// TwinCAT 3 PLC project TwinCore
// Title: TwinCore
// Company: TwinCore
// Author: TwinCore
// ProjectVersion: 2026.24.1.0
// Description: base implementations, utilities, TC3 event logging, state machines, ...
// ProgramVersion: 3.1.4026.23
// libraries:
//   Tc2_Standard, * (Beckhoff Automation GmbH)
//   Tc2_System, * (Beckhoff Automation GmbH)
//   Tc2_Utilities, * (Beckhoff Automation GmbH)
//   Tc3_EventLogger, * (Beckhoff Automation GmbH)
//   Tc3_Module, * (Beckhoff Automation GmbH)
// project tree:
//   EventLogger/EventListenerExtV2/DUTs/ E_AlarmMessage.TcDUT, ST_AlarmInfo.TcDUT, ST_AlarmLog.TcDUT, ST_EventEntryTableListener.TcDUT
//   EventLogger/EventListenerExtV2/ FB_EventListenerExtV2.TcPOU, I_EventListener.TcIO
//   EventLogger/EventManagement/DUTs/ E_AlarmReaction.TcDUT, ST_EventEntryTable.TcDUT, ST_EventHmiControl.TcDUT
//   EventLogger/EventManagement/ FB_Alarm.TcPOU, FB_AlarmDelayed.TcPOU, FB_AlarmManagement.TcPOU, FB_Message.TcPOU, I_Alarm.TcIO, I_Message.TcIO
//   EventLogger/Logger/ E_RollingInterval.TcDUT, FB_FileRetentionTimeHandler.TcPOU, FB_GenerateTimeData.TcPOU, FB_Log.TcPOU, FB_LogFile.TcPOU, FB_LogStringBuffer.TcPOU, FB_SystemTimeService.TcPOU, F_GetFileAgeInSeconds.TcPOU, ST_LogEntry.TcDUT
//   General/Blinker/ FB_Blinker.TcPOU, FB_Blinker_PWM.TcPOU
//   General/CONCAT/ FB_CONCAT.TcPOU, FB_CONCAT_STRINGS.TcPOU, I_CONCAT.TcIO
//   General/ FB_AnalogInputFilter.TcPOU, FB_Signal.TcPOU
//   GVLs/ GVL_Diag.TcGVL, GVL_GLOBAL.TcGVL
//   Lists/ FB_ListNumbers_DINT.TcPOU, FB_ListNumbers_REAL.TcPOU, FB_ListString.TcPOU
//   Misc/ ST_LinCoord_XY.TcDUT, ST_LinCoord_XYZ.TcDUT, ST_SysTime.TcDUT
//   / Parameter.TcGVL
//   Process/DUTs/ ST_Position.TcDUT, ST_ProcessData.TcDUT, ST_Task.TcDUT
//   Process/ FB_Process.TcPOU
//   Project Information/ F_GetCompany.TcPOU, F_GetTitle.TcPOU, F_GetVersion.TcPOU
//   StateMachine/ FB_StateMachine.TcPOU, ST_HMI_Condition.TcDUT, ST_HMI_StateMachine.TcDUT, ST_StateMachine_State.TcDUT
//   StateMachine/MachineState/ E_MachineState.TcDUT, FB_MachineState.TcPOU, ST_MachineInfo.TcDUT
//   StateMachine/ModeControl/ E_Mode.TcDUT, FB_ModeControl.TcPOU
//   Version/ Global_Version.TcGVL

// ---- EventLogger/EventListenerExtV2/DUTs/E_AlarmMessage.TcDUT
{attribute 'qualified_only'}
{attribute 'strict'}
TYPE E_AlarmMessage :
(
	RequestText := 0,
    ReceiveText := 1,
    Insert := 2,
    WriteDB := 3,
    Done := 4
);
END_TYPE

// ---- EventLogger/EventListenerExtV2/DUTs/ST_AlarmInfo.TcDUT
TYPE ST_AlarmInfo :
STRUCT
	bVerbose: BOOL;
	nVerboseRaisedCount: UDINT;
	bInfo: BOOL;
	nInfoRaisedCount: UDINT; 
	bWarning: BOOL;
	nWarningRaisedCount: UDINT;
	bError: BOOL;
	nErrorRaisedCount: UDINT;
	bCritical: BOOL;
	nCriticalRaisedCount: UDINT;
END_STRUCT
END_TYPE

// ---- EventLogger/EventListenerExtV2/DUTs/ST_AlarmLog.TcDUT
TYPE ST_AlarmLog :
STRUCT
	sTimestamp: STRING;
	sText: STRING(255); //
	sSourceName: STRING(255); //
	EventClassName: STRING(255); //
    eConfirmationState : INT;
    eSeverity :  INT; // INT
END_STRUCT
END_TYPE

// ---- EventLogger/EventListenerExtV2/DUTs/ST_EventEntryTableListener.TcDUT
TYPE ST_EventEntryTableListener EXTENDS ST_EventEntryTable:
STRUCT
	sJsonAttribute	: STRING(8000);
	ipArguments		: I_TcArguments;
END_STRUCT
END_TYPE

// ---- EventLogger/EventManagement/DUTs/E_AlarmReaction.TcDUT
{attribute 'qualified_only'}
{attribute 'strict'}
TYPE E_AlarmReaction :
(
	None := 0,
	Info,
	Warning,
	Verbose,
	StopAtCycleEnd,
	AbortGroup,
	AbortAll,
	MediaOff
);
END_TYPE

// ---- EventLogger/EventManagement/DUTs/ST_EventEntryTable.TcDUT
TYPE ST_EventEntryTable EXTENDS ST_LogEntry :
STRUCT
	nSourceId			: UDINT;
	nZoneId				: UDINT;
	nGroupId			: UDINT;
	sDescription		: T_MaxString;
	eSeverity			: TcEventSeverity;
	eReaction			: E_AlarmReaction;
    sReaction			: STRING( 24 );
	EventClass			: GUID;
	EventClassName		: T_MaxString;
	sTimestamp			: STRING( 24 );
	sTimestampConfirmed	: STRING( 24 );
	sTimestampCleared	: STRING( 24 );
	nEventId			: UDINT;
	eConfirmationState	: TcEventConfirmationState;
	bTextRecieved		: BOOL;
	bIsAlarm			: BOOL;
	bIsEvent			: BOOL;
    stAlarmLog			: ST_AlarmLog;
    bLogged				: BOOL;
    nLanguageId			: INT;
END_STRUCT
END_TYPE

// ---- EventLogger/EventManagement/DUTs/ST_EventHmiControl.TcDUT
TYPE ST_EventHmiControl :
STRUCT
END_STRUCT
END_TYPE

// ---- EventLogger/Logger/E_RollingInterval.TcDUT
{attribute 'qualified_only'}
{attribute 'strict'}
{attrivute 'to_string'}
// Rolling interval to create a new log file when expired. 
TYPE E_RollingInterval : (
    None,
    Hourly,
    Daily,
    Monthly
);
END_TYPE

// ---- EventLogger/Logger/ST_LogEntry.TcDUT
TYPE ST_LogEntry :
STRUCT
	sSeverity		:  STRING( 24 );
	sSourceName		: T_MaxString;
	sTimestampLog	: STRING( 24 );
	MethodName		: STRING( 24 );
	sText			: T_MaxString;
END_STRUCT
END_TYPE

// ---- Misc/ST_LinCoord_XY.TcDUT
TYPE ST_LinCoord_XY :
STRUCT
	x	: REAL;	// [mm]
	y	: REAL;	// [mm]
END_STRUCT
END_TYPE

// ---- Misc/ST_LinCoord_XYZ.TcDUT
TYPE ST_LinCoord_XYZ EXTENDS ST_LinCoord_XY :
STRUCT
	z	: REAL;	// [mm]
END_STRUCT
END_TYPE

// ---- Misc/ST_SysTime.TcDUT
TYPE ST_SysTime :
STRUCT
	uliDateTime	: ULINT := 0;
	sTimestamp	: STRING(12); // current time, format: hh:mm:ss:ms
	sDate		: STRING(10); // current date, format example: dd.mm.yyyy
	uiYear		: UINT := 0;
	uiMonth		: UINT := 9999;
	uiDay		: UINT := 9999;
	uiHour		: UINT := 9999;
	uiMinute	: UINT := 9999;
	uiSecond	: UINT := 9999;
	uiMillis	: UINT := 9999;
END_STRUCT
END_TYPE

// ---- Process/DUTs/ST_Position.TcDUT
TYPE ST_Position :
STRUCT
	Task		: ARRAY[0..Parameter.MAX_TASK_INDEX] OF ST_Task;
	Group		: ARRAY[0..Parameter.MAX_GROUP_INDEX] OF ST_Task;
	Info		: ST_Task;
END_STRUCT
END_TYPE

// ---- Process/DUTs/ST_ProcessData.TcDUT
TYPE ST_ProcessData :
STRUCT
	Pos	: ARRAY[0..Parameter.MAX_POS_INDEX] OF ST_Position;
	Info		: ST_Task;	// info about the complete process of all positions
END_STRUCT
END_TYPE

// ---- Process/DUTs/ST_Task.TcDUT
TYPE ST_Task :
STRUCT
	Enabled		: BOOL := FALSE;	// false if not existing
	Released	: BOOL;	// free to start this task
	Busy		: BOOL;	// task started
	Finished	: BOOL;	// also TRUE, when all Tasks are disabled
	OK			: BOOL;
	NOK			: BOOL;
	ManualOK	: BOOL;
	ManualNOK	: BOOL;
	State		: USINT;	// lamp HMI
	(*	State
		0 - not existing
		1 - existing/enabled, but not released
		2 - enabled and released, ready to process
		3 - processing, process started
		4 - OK
		5 - NOK
		6 - ManualOK
		7 - ManualNOK
	*)
	_groupID	: USINT := 0;
END_STRUCT
END_TYPE

// ---- StateMachine/MachineState/E_MachineState.TcDUT
{attribute 'qualified_only'}
TYPE E_MachineState :
(
	Error := -1,
	Idle := 0,
	Stopped,	// Manual Control
	Stopping,
	Aborting,
	Aborted,
	Starting,
	Execute,	// Automatic
	Hold,
	Homing,
	Clearing,
	Resetting
);
END_TYPE

// ---- StateMachine/MachineState/ST_MachineInfo.TcDUT
TYPE ST_MachineInfo :
STRUCT
	bInInitDone:	BOOL;
	bInMediaOn:		BOOL;
END_STRUCT
END_TYPE

// ---- StateMachine/ModeControl/E_Mode.TcDUT
{attribute 'qualified_only'}
TYPE E_Mode :
(
	Error := -1,
	Idle := 0,
	Stopped,	// Manual Control
	Stopping,
	Aborting,
	Aborted,
	Starting,
	Hold,
	Homing,
	Clearing,
	Resetting,
	Standby,	// Automatic
	Execute	// Automatic
);
END_TYPE

// ---- StateMachine/ST_HMI_Condition.TcDUT
TYPE ST_HMI_Condition :
STRUCT
	xState	: BOOL := TRUE;
	sName	: STRING(26) := '';
END_STRUCT
END_TYPE

// ---- StateMachine/ST_HMI_StateMachine.TcDUT
TYPE ST_HMI_StateMachine :
STRUCT
	// name of state machine
	sName				: STRING;	

	// current state
	nState				: INT;
	nNextState			: INT;	// prepared next state
	sState				: STRING;
	
	// conditions
	stSwitchCondition	: ARRAY[0..Parameter.NUM_CON] OF ST_HMI_Condition;
	stStateCondition	: ARRAY[0..Parameter.NUM_CON] OF ST_HMI_Condition;
	
	nSwitchOrSection	: INT;	// current or section
	bShowOrSection		: BOOL;	// show or section elements
	bShowNextState		: BOOL;	// show next state
	bSwitchOrSectionDec	: BOOL;	// decrement
	bSwitchOrSectionInc	: BOOL;	// increment
	bStepMode			: BOOL;
	bStepNext			: BOOL;
	
	// Log
	stStateHistory		: ARRAY[0..Parameter.HISTORY_SIZE] OF ST_StateMachine_State;
END_STRUCT
END_TYPE

// ---- StateMachine/ST_StateMachine_State.TcDUT
TYPE ST_StateMachine_State :
STRUCT
	nState	: INT;
	sState	: STRING;
END_STRUCT
END_TYPE

// ---- GVLs/GVL_Diag.TcGVL
{attribute 'qualified_only'}
VAR_GLOBAL
	gfbAlarmManagement			: FB_AlarmManagement;	// first: nested FB_Alarm.FB_init prepends onto ipAlarmHead
	gfbLogFile					: FB_LogFile;
	gfbEventListener			: FB_EventListenerExtV2; // other HMI than TE2000
	ipAlarmHead					: I_Alarm;	// singly linked list of all FB_Alarm instances
	gnCountAlarms				: UINT := 0;	// built-in and user FB_Alarm instances self-register in FB_init
	gbCountAlarmsMaxExceeded	: BOOL := FALSE;
	gbInterfaceNotAssigned		: BOOL := FALSE;
	
END_VAR

// ---- GVLs/GVL_GLOBAL.TcGVL
{attribute 'Tc2GvlVarNames'}
VAR_GLOBAL
	fbConcat		: FB_CONCAT;
    fbSystemTime	: FB_SystemTimeService;
END_VAR

// ---- Parameter.TcGVL
{attribute 'qualified_only'}
VAR_GLOBAL CONSTANT
	
    MAX_STRING_LENGTH	: UDINT := 255;
	
	
	// Alarm Management
	nMaxNumberAlarms		: UINT := 2000;	// safety cap for FB_Alarm linked-list registration (not an array size)
	
	// Logger
	MAX_LOG_STRING_SIZE		: UINT := 1000;	// maximal string size for one log entry (line)
    MAX_BUFFER_COUNT		: UDINT := 1000;
	
	// Following for other HMI solution than TE2000
	nMaxEventEntries		: UINT := 200;	// max. event entries in EventEntryTable
	
	// Listener
	nMaxEventClasses		: UINT := 2;	// Listener - max. event classes
	nNUM_OF_MESSAGES_VISU	: UINT := 15;	// Listener - messages to store and read from HMI
	
	
	// state machine
	NUM_CON			: USINT := 15;
	HISTORY_SIZE	: INT := 30;
	
	// Process
	MAX_POS_INDEX	: INT := 4;
	MAX_TASK_INDEX	: INT := 81;
	MAX_GROUP_INDEX	: INT := 15;
	
END_VAR

// ---- Version/Global_Version.TcGVL
{attribute 'TcGenerated'}
{attribute 'no-analysis'}
{attribute 'linkalways'}
// This function has been automatically generated from the project information.
VAR_GLOBAL CONSTANT
	{attribute 'const_non_replaced'}
	stLibVersion_TwinCore : ST_LibVersion := (iMajor := 2026, iMinor := 24, iBuild := 1, iRevision := 0, nFlags := 1, sVersion := '2026.24.1.0');
END_VAR

// ---- EventLogger/EventListenerExtV2/I_EventListener.TcIO
INTERFACE I_EventListener EXTENDS __SYSTEM.IQueryInterface

METHOD PUBLIC DeleteEventsFromTable : BOOL
END_METHOD

METHOD GetEventByIndex : HRESULT
    VAR_OUTPUT
        sTimestamp: STRING(80); // 
        sTimestampConfirmed: STRING(80);
        sTimestampCleared: STRING(80);
        sText: STRING(255); //
        sSourceName: STRING(255); //
        EventClassName: STRING(255); //
        eConfirmationState : BYTE;
        eSeverity :  BYTE; // INT
    END_VAR
VAR_INPUT
    nIndex : UDINT;
END_VAR
END_METHOD

PROPERTY PUBLIC LangId : INT
GET
END_GET
SET
END_SET
END_PROPERTY

PROPERTY NumberActiveEvents : UDINT
GET
END_GET
END_PROPERTY

END_INTERFACE

// ---- EventLogger/EventManagement/I_Alarm.TcIO
INTERFACE I_Alarm EXTENDS I_Message

METHOD Ack : HRESULT
VAR_INPUT
END_VAR
END_METHOD

PROPERTY bActive : BOOL
GET
END_GET
END_PROPERTY

PROPERTY PUBLIC bBlockAck : BOOL
GET
END_GET
SET
END_SET
END_PROPERTY

PROPERTY bRaised : BOOL
GET
END_GET
END_PROPERTY

PROPERTY PUBLIC eEventReaction : E_AlarmReaction
GET
END_GET
END_PROPERTY

PROPERTY ipNext : I_Alarm
GET
END_GET
SET
END_SET
END_PROPERTY

METHOD PUBLIC UpdateText : HRESULT
VAR_INPUT
	LangId	: INT;
END_VAR
END_METHOD

END_INTERFACE

// ---- EventLogger/EventManagement/I_Message.TcIO
 INTERFACE I_Message

PROPERTY PUBLIC bSetEvent : BOOL
GET
END_GET
SET
END_SET
END_PROPERTY

PROPERTY eSeverity : TcEventSeverity
GET
END_GET
END_PROPERTY

METHOD GetEventEntry : ST_EventEntryTable
VAR_INPUT
END_VAR
END_METHOD

METHOD GetEventText : BOOL
VAR_INPUT
END_VAR
END_METHOD

METHOD GetJsonAttribute : HRESULT
VAR_INPUT
	sJsonAttribute	: REFERENCE TO STRING;
	nJsonAttribute	: UDINT;
END_VAR
END_METHOD

PROPERTY PUBLIC LogEntry : ST_LogEntry
GET
END_GET
END_PROPERTY

PROPERTY PUBLIC nGetGroupId : UINT
GET
END_GET
END_PROPERTY

PROPERTY PUBLIC nGetSourceId : UDINT
GET
END_GET
END_PROPERTY

END_INTERFACE

// ---- General/CONCAT/I_CONCAT.TcIO
INTERFACE I_CONCAT

METHOD AddString : I_CONCAT
VAR_INPUT
	pSrcString	: ANY_STRING;
END_VAR
END_METHOD

METHOD AddStringInput : I_CONCAT
VAR_INPUT
	in:	STRING;
END_VAR
END_METHOD

METHOD PUBLIC Get : T_MAXSTRING
VAR_INPUT
END_VAR
END_METHOD

END_INTERFACE

// ---- EventLogger/EventManagement/FB_AlarmManagement.TcPOU
FUNCTION_BLOCK FB_AlarmManagement
VAR_INPUT
	bInAck			: BOOL;	// Acknowledge all errors, if possible
END_VAR
VAR_OUTPUT
	bError			: BOOL;	// Alarm active with reaction type media off or abort all
	
	// MessageReaction
	bVerbose		: BOOL;	// at least one verbose info is active (not important info)
	bInfo			: BOOL;	// at least one info is active
	bWarning		: BOOL;	// at least one warning is active
	bStopAtCycleEnd	: BOOL;	// at least on alarm needs to stop at cycle end, goes into stop state after ending cycle
	bAbortGroup		: BOOL;	// aborts one group, detect with method IsAlarmInGroup( GroupID ) or IsAlarmInGroupOfZone( GroupID )
	bAbortAll		: BOOL;	// abort/stops all groups
	bMediaOff		: BOOL;	// critical alarm, shuts down media!
	
	bAckRequested	: BOOL;	// at least one verbose info is active (not important info)
	
    aEventEntryTable: ARRAY[0..Parameter.nMaxEventEntries] OF ST_EventEntryTable;	// to show in HMI
	
END_VAR
VAR
	bInit	: BOOL := TRUE;
	
    nCounter	: UINT;

	rtAck	: R_TRIG;
	
	nVisuTableIndex					: UINT;
	bVisuTableCmdIndexPlus			: BOOL;
	bVisuTableCmdIndexMinus			: BOOL;
	bVisuTableDisableCmdIndexPlus	: BOOL;
	bVisuTableDisableCmdIndexMinus	: BOOL;
	bVisuTableCmdCleanErrors		: BOOL;
	
    nLanguage	: INT := 1031;
    sLanguage	: STRING := 'de';
    bChangeLanguage	: BOOL;
	
	cfgShowErrors	: BOOL := TRUE;	// including critical
	cfgShowWarnings	: BOOL := TRUE;
	cfgShowInfos	: BOOL := TRUE;	// including verbose
	
    fbSourceInfo				: FB_TcSourceInfo;
    fbGetTimeZoneInformation	: FB_GetTimeZoneInformation;
    stSeverestAlarmEntryTable	: ST_EventEntryTable;
    stLastEventEntryTable		: ST_EventEntryTable;
	
	fbWrnTooManyAlarms			: FB_Alarm( TC_EVENTS.EventClassGeneral.W_TooManyAlarmsDefined );
	fbErrInterfaceNotAssigned	: FB_Alarm( TC_EVENTS.EventClassGeneral.E_Debug );
	fbWrnArgumentBeforeInit		: FB_Alarm( TC_EVENTS.EventClassGeneral.W_ArgumentBeforeInit );
	fbWrnCyclicCallNotDetected	: FB_Alarm( TC_EVENTS.EventClassGeneral.W_CyclicCallNotDetected );
	{warning 'TODO: realize cyclic call detection'}
	
END_VAR


// in case you only want to call the body cyclic.
Execute( bInAck );

{warning 'TODO: log history of general events! Verbose/Debug'}

// cyclic call of Event Management, in case you don't want to use the FB-body!
METHOD PUBLIC Execute : HRESULT
VAR_INPUT
	bInAck			: BOOL;	// Acknowledge all errors, if possible
END_VAR
VAR_INST
    bGetTimeZone : BOOL := TRUE;
END_VAR

// inititalizing
IF bInit THEN
	Initialize();
END_IF

// trigger of inputs
rtAck( CLK := bInAck OR bVisuTableCmdCleanErrors );
bVisuTableCmdCleanErrors R= bVisuTableCmdCleanErrors;

// check if at least one Error is raised, and store alarm reaction type
initOutputs();

// Update Language
LanguageId( sLanguage );

// Update event table
UpdateEventTable();

// HMI
HMI();

fbGetTimeZoneInformation( bExecute := bGetTimeZone );
bGetTimeZone R= bGetTimeZone;

// Debug Meldungen 
fbWrnTooManyAlarms.setEvent( GVL_Diag.gbCountAlarmsMaxExceeded );
fbErrInterfaceNotAssigned.setEvent( GVL_Diag.gbInterfaceNotAssigned );
fbWrnArgumentBeforeInit.setEvent( FALSE );
END_METHOD

METHOD FB_exit : BOOL
VAR_INPUT
	bInCopyCode : BOOL; // if TRUE, the exit method is called for exiting an instance that is copied afterwards (online change).
END_VAR

IF NOT bInCopyCode THEN
	; // each nested FB_Alarm.FB_exit unlinks itself from ipAlarmHead
END_IF
END_METHOD

METHOD PUBLIC GetEventTable : BOOL
VAR_INPUT
	nZoneId		: UDINT;	// Zone = 0 is for all zones
	nGroupId	: UINT;
	bShowError	: BOOL;	// including criticals
	bShowWarning: BOOL;
	bShowInfo	: BOOL;	// including verbose
END_VAR
VAR_IN_OUT
	astEventTable	:	ARRAY[*] OF ST_EventEntryTable;
END_VAR
VAR
	i			: DINT;
	j			: DINT;
	nLowerBound	: DINT;
	nUpperBound	: DINT;
	EmptyEventTableLine	: ST_EventEntryTable;
END_VAR

// check bounds
nLowerBound := LOWER_BOUND( astEventTable, 1 );
nUpperBound := UPPER_BOUND( astEventTable, 1 );
j := nLowerBound;

// empty table
FOR i := nLowerBound TO nUpperBound DO	
	astEventTable[i] := EmptyEventTableLine;
END_FOR

// poll the big Event table
FOR i := 0 TO Parameter.nMaxEventEntries DO

	// check filter settings
	IF ( nZoneId <> 0 AND aEventEntryTable[i].nZoneId = nZoneId )
	OR_ELSE ( nGroupId <> 0 AND aEventEntryTable[i].nGroupId = nGroupId )
	AND_THEN ( ( aEventEntryTable[i].eSeverity = TcEventSeverity.Critical AND bShowError )
		OR ( aEventEntryTable[i].eSeverity = TcEventSeverity.Error AND bShowError )
		OR ( aEventEntryTable[i].eSeverity = TcEventSeverity.Warning AND bShowWarning )
		OR ( aEventEntryTable[i].eSeverity = TcEventSeverity.Info AND bShowInfo )
		OR ( aEventEntryTable[i].eSeverity = TcEventSeverity.Verbose AND bShowInfo ) )
	THEN
		
		// fill filtered feedback table
		astEventTable[j] := aEventEntryTable[i];
		j := j + 1;
		
	END_IF
	
	// used table is full
	IF j > nUpperBound THEN
		RETURN;
	END_IF
	
END_FOR
END_METHOD

METHOD PRIVATE HMI : BOOL
VAR_INST
    nCounterTemp : DINT;
    trigVisuIndexingPlus: R_TRIG;
	trigVisuIndexingMinus: R_TRIG;
END_VAR

IF nCounterTemp <> nCounter THEN
    nCounterTemp := nCounter;
    nVisuTableIndex := 0;
END_IF

bVisuTableDisableCmdIndexPlus := nVisuTableIndex > nCounter - Parameter.nNUM_OF_MESSAGES_VISU
	OR nCounter <= Parameter.nNUM_OF_MESSAGES_VISU
	OR nVisuTableIndex >= Parameter.nMaxEventEntries;

bVisuTableDisableCmdIndexMinus := nVisuTableIndex <= 0;

trigVisuIndexingPlus( CLK := bVisuTableCmdIndexPlus );
IF trigVisuIndexingPlus.Q THEN
	nVisuTableIndex := nVisuTableIndex + 1;
END_IF

trigVisuIndexingMinus( CLK := bVisuTableCmdIndexMinus );
IF trigVisuIndexingMinus.Q THEN
	nVisuTableIndex := nVisuTableIndex - 1;
END_IF
END_METHOD

METHOD PRIVATE Initialize : BOOL
VAR_INPUT
END_VAR

fbWrnTooManyAlarms.Initialize( 0, 0, E_AlarmReaction.Warning );
fbErrInterfaceNotAssigned.Initialize( 0, 0, E_AlarmReaction.AbortAll );
fbWrnArgumentBeforeInit.Initialize( 0, 0, E_AlarmReaction.Warning );

bInit := FALSE;
END_METHOD

METHOD PRIVATE initOutputs : BOOL
VAR_INPUT
END_VAR

bError			:= FALSE;
bInfo			:= FALSE;
bWarning		:= FALSE;
bVerbose		:= FALSE;
bStopAtCycleEnd	:= FALSE;
bAbortGroup		:= FALSE;
bAbortAll		:= FALSE;
bMediaOff		:= FALSE;
END_METHOD

METHOD PUBLIC IsAlarmInGroup : BOOL
VAR_INPUT
	nGroupId	: UINT;
END_VAR
VAR
	ipAlarm	: I_Alarm;
	nGuard	: UINT;
END_VAR

IsAlarmInGroup := FALSE;
ipAlarm := GVL_Diag.ipAlarmHead;
nGuard := 0;
WHILE ipAlarm <> 0 AND nGuard < Parameter.nMaxNumberAlarms DO
	nGuard := nGuard + 1;
	IF ipAlarm.bActive
	AND_THEN ipAlarm.nGetGroupId = nGroupId THEN
		IsAlarmInGroup := TRUE;
		RETURN;
	END_IF
	ipAlarm := ipAlarm.ipNext;
END_WHILE
END_METHOD

METHOD PUBLIC IsAlarmInGroupOfZone : BOOL
VAR_INPUT
	nZoneId		: UDINT;
	nGroupId	: UINT;
END_VAR
VAR
	ipAlarm	: I_Alarm;
	nGuard	: UINT;
END_VAR

IsAlarmInGroupOfZone := FALSE;
ipAlarm := GVL_Diag.ipAlarmHead;
nGuard := 0;
WHILE ipAlarm <> 0 AND nGuard < Parameter.nMaxNumberAlarms DO
	nGuard := nGuard + 1;
	IF ipAlarm.bActive
	AND_THEN ipAlarm.nGetGroupId = nGroupId
	AND ipAlarm.nGetSourceId = nZoneId THEN
		IsAlarmInGroupOfZone := TRUE;
		RETURN;
	END_IF
	ipAlarm := ipAlarm.ipNext;
END_WHILE
END_METHOD

METHOD PUBLIC IsAlarmInZone : BOOL
VAR_INPUT
	nZoneId	: UDINT;
END_VAR
VAR
	ipAlarm	: I_Alarm;
	nGuard	: UINT;
END_VAR

IsAlarmInZone := FALSE;
ipAlarm := GVL_Diag.ipAlarmHead;
nGuard := 0;
WHILE ipAlarm <> 0 AND nGuard < Parameter.nMaxNumberAlarms DO
	nGuard := nGuard + 1;
	IF ipAlarm.bActive
	AND_THEN ipAlarm.nGetSourceId = nZoneId THEN
		IsAlarmInZone := TRUE;
		RETURN;
	END_IF
	ipAlarm := ipAlarm.ipNext;
END_WHILE
END_METHOD

METHOD PUBLIC LanguageId : HRESULT
VAR_INPUT
	sCurrentLanguage	: STRING;
END_VAR
VAR
	ipAlarm	: I_Alarm;
	nGuard	: UINT;
	hrChangeLang	:HRESULT;
	bChangeLangPending	:BOOL;
	bChangeLangSuccess	:BOOL;
	bChangeLangError	:BOOL;
END_VAR

// Set language
IF sLanguage <> sCurrentLanguage THEN
	IF sCurrentLanguage = 'de' OR sCurrentLanguage = 'DE' THEN
		nLanguage := 1031;
	ELSIF sCurrentLanguage = 'en' OR sCurrentLanguage = 'EN' OR sCurrentLanguage = 'gb' OR sCurrentLanguage = 'GB' THEN
		nLanguage := 1033;
	ELSIF sCurrentLanguage = 'cz' OR sCurrentLanguage = 'CZ' THEN
		nLanguage := 1029;
	END_IF
	
	sLanguage := sCurrentLanguage;
	bChangeLanguage := TRUE;
END_IF

{warning 'TODO: Sprachenänderung realisieren'}
IF bChangeLanguage AND FALSE THEN
	// update text
	
	bChangeLangPending := FALSE;
	bChangeLangSuccess := TRUE;
	bChangeLangError := FALSE;
	ipAlarm := GVL_Diag.ipAlarmHead;
	nGuard := 0;
	WHILE ipAlarm <> 0 AND nGuard < Parameter.nMaxNumberAlarms DO
		nGuard := nGuard + 1;
		hrChangeLang := ipAlarm.UpdateText( nLanguage );
		IF hrChangeLang = S_PENDING THEN
			bChangeLangPending := TRUE;
		END_IF
		IF hrChangeLang = E_FAIL THEN
			bChangeLangError := TRUE;
		END_IF
		IF hrChangeLang <> S_OK THEN
			bChangeLangSuccess := FALSE;
		END_IF
		ipAlarm := ipAlarm.ipNext;
	END_WHILE
	
	IF bChangeLangSuccess THEN
		bChangeLanguage := FALSE;
	END_IF
	
END_IF
END_METHOD

METHOD PRIVATE UpdateEventTable : BOOL
VAR_INPUT
END_VAR
VAR
	ipAlarm	: I_Alarm;
	j		: UINT;
	nGuard	: UINT;
END_VAR
VAR_INST
    stEventEntryTemp: ST_EventEntryTable;
END_VAR

// Init output table
MEMSET( ADR( aEventEntryTable ), 0, SIZEOF( aEventEntryTable ) );
j := 0;
bAckRequested := FALSE;

ipAlarm := GVL_Diag.ipAlarmHead;
nGuard := 0;
WHILE ipAlarm <> 0 AND nGuard < Parameter.nMaxNumberAlarms DO
	nGuard := nGuard + 1;
	
	// alarm is active
	IF ipAlarm.bActive THEN
		
		// Acknowledge errors
		IF rtAck.Q THEN
			ipAlarm.Ack();
		END_IF
		
		// reset _bSetEvent to check, if it will be set again
		IF NOT ipAlarm.bSetEvent THEN
			ipAlarm.bBlockAck := FALSE;
		END_IF
		ipAlarm.bSetEvent := FALSE;
		
		// if there is at least one acknowledgable alarm
		bAckRequested S= NOT ipAlarm.bBlockAck AND ipAlarm.bActive;
		
		// update text
		ipAlarm.UpdateText( nLanguage );
		
		// fill table for HMI
		IF j <= Parameter.nMaxEventEntries
		AND_THEN ( ( ipAlarm.eSeverity = TcEventSeverity.Critical AND cfgShowErrors )
			OR ( ipAlarm.eSeverity = TcEventSeverity.Error AND cfgShowErrors )
			OR ( ipAlarm.eSeverity = TcEventSeverity.Warning AND cfgShowWarnings )
			OR ( ipAlarm.eSeverity = TcEventSeverity.Info AND cfgShowInfos )
			OR ( ipAlarm.eSeverity = TcEventSeverity.Verbose AND cfgShowInfos ) )
		THEN
			aEventEntryTable[j] := ipAlarm.GetEventEntry();
			aEventEntryTable[j].bIsAlarm := TRUE;
			j := j + 1;
		END_IF
		
		// alarm reactions
		CASE ipAlarm.eEventReaction OF
			E_AlarmReaction.None:
				;
			E_AlarmReaction.Info:
				bInfo := TRUE;
			E_AlarmReaction.Warning:
				bWarning := TRUE;
			E_AlarmReaction.Verbose:
				bVerbose := TRUE;
			E_AlarmReaction.StopAtCycleEnd:
				bStopAtCycleEnd := TRUE;
			E_AlarmReaction.AbortGroup:
				bAbortGroup := TRUE;
				bError := TRUE;
			E_AlarmReaction.AbortAll:
				bAbortAll := TRUE;
				bError := TRUE;
			E_AlarmReaction.MediaOff:
				bMediaOff := TRUE;
				bError := TRUE;
		ELSE
			;
		END_CASE

		// severity critical is dominant
		bError S= ipAlarm.eSeverity = TcEventSeverity.Critical;
		
	END_IF
	
	ipAlarm := ipAlarm.ipNext;
END_WHILE
END_METHOD

METHOD PRIVATE UpdateLegacyTable : ARRAY[1..80] OF ST_ReadEvent
VAR_INPUT
END_VAR
VAR
	i	: UINT;
END_VAR

// Init output table
MEMSET(ADR(UpdateLegacyTable),0,SIZEOF(UpdateLegacyTable));

FOR i := 1 TO MIN( 80, Parameter.nMaxEventEntries + 1 ) BY 1 DO
	
	// Severity
	CASE aEventEntryTable[i-1].eSeverity OF 
		TcEventSeverity.Verbose :
			UpdateLegacyTable[i].nClass := 0;
		TcEventSeverity.Info :
			UpdateLegacyTable[i].nClass := 4;
		TcEventSeverity.Warning :
			UpdateLegacyTable[i].nClass := 6; 
		TcEventSeverity.Error :
			UpdateLegacyTable[i].nClass := 7;
		TcEventSeverity.Critical :
			UpdateLegacyTable[i].nClass := 7;  
	END_CASE
	
	// state of confirmation and reset
	 CASE aEventEntryTable[i-1].eConfirmationState OF 
		TcEventConfirmationState.NotSupported :
			UpdateLegacyTable[i].nConfirmState := 0;
			UpdateLegacyTable[i].nResetState := 0;
			
		TcEventConfirmationState.NotRequired :
			UpdateLegacyTable[i].nConfirmState := 3;
			UpdateLegacyTable[i].nResetState := 0;
			
		TcEventConfirmationState.WaitForConfirmation :
			UpdateLegacyTable[i].nConfirmState := 1;
			UpdateLegacyTable[i].nResetState := 1;

		TcEventConfirmationState.Confirmed :
			UpdateLegacyTable[i].nConfirmState := 4;
			UpdateLegacyTable[i].nResetState := 3;
			
		TcEventConfirmationState.Reset :
			UpdateLegacyTable[i].nConfirmState := 0;
			UpdateLegacyTable[i].nResetState := 3;  
	END_CASE
				
	// rest of data
	UpdateLegacyTable[i].nEventId := aEventEntryTable[i-1].nEventId;
	UpdateLegacyTable[i].sComputer := aEventEntryTable[i-1].EventClassName;
	UpdateLegacyTable[i].sDate := LEFT( aEventEntryTable[i-1].sTimestamp, 10 );
	UpdateLegacyTable[i].sMessageText := aEventEntryTable[i-1].sText;
	UpdateLegacyTable[i].sSource := aEventEntryTable[i-1].sSourceName;
	UpdateLegacyTable[i].nSourceId := aEventEntryTable[i-1].nSourceId;
	UpdateLegacyTable[i].sTime := LEFT( DELETE( aEventEntryTable[i-1].sTimestamp, 11, 1 ), 8 );
	
END_FOR
END_METHOD

END_FUNCTION_BLOCK

// ---- EventLogger/EventManagement/FB_Alarm.TcPOU
//Usage description
//-----------------
//| This FB uses the FB_init, which needs to be initialized within the declaration!
//| Also it can use the method Initialization, to specify Group/Zone IDs of the Event. Here you can also change the alarm reaction
//| FB_init / Initialize prepend this instance onto GVL_Diag.ipAlarmHead (linked list, no GVL table).
//| use SetEvent[...] -methods to raise an alarm!
//| 
//| You can trigger an alarm once or use it cyclically.
//| The :ref:`FB_AlarmManagement` prevent acknowledge automatically if SetAlarm is still set.
FUNCTION_BLOCK FB_Alarm IMPLEMENTS I_Alarm
VAR_INPUT
END_VAR
VAR_OUTPUT
	sText		: STRING := '';
	sClassName	: STRING := '';
	sTimeRaised	: STRING := '';
	nGroupId	: UINT;
	nZoneId		: UINT;
END_VAR
VAR
	_bSetEvent				: BOOL;
	_bBlockAck				: BOOL;
	_bWithConfirmation		: BOOL;
	fbTcAlarm				: FB_TcAlarm;
	_fbInternalSourceInfo	: Tc3_EventLogger.FB_TcSourceInfo;	// needed to have "multi-instances" of EventClass in CreateEx()
	nLangId					: INT;
	
    fbRequestText : FB_RequestEventText;
    fbRequestClassName : FB_RequestEventClassName;
	
	_stEventClass	: TcEventEntry;
	_eEventReaction	: E_AlarmReaction;
	_ipNext			: I_Alarm;
	_nArgumentCount: UDINT;
	
	hrRaise	: HRESULT;
END_VAR

METHOD Ack : HRESULT
VAR_INPUT
END_VAR

IF NOT _bBlockAck AND_THEN THIS^.bActive THEN
	Ack := THIS^.fbTcAlarm.Clear( 0, FALSE );
ELSE
	Ack := 1;
END_IF
END_METHOD

METHOD PUBLIC AddArgument : REFERENCE TO FB_Alarm
VAR_INPUT
	sName	: STRING;
END_VAR

THIS^.fbTcAlarm.ipArguments.AddString( sName );
addArgument REF= THIS^;
_nArgumentCount := _nArgumentCount + 1;
END_METHOD

// Returns TRUE if the alarm is in the "Raised" or "Wait For Confirmation" state.
PROPERTY bActive : BOOL
GET
bActive := THIS^.fbTcAlarm.bActive OR _bSetEvent;
END_GET
END_PROPERTY

PROPERTY PUBLIC bBlockAck : BOOL
GET
bBlockAck := _bBlockAck;
END_GET
SET
_bBlockAck := bBlockAck;
END_SET
END_PROPERTY

// Returns TRUE if the alarm is in the "raised" state.
PROPERTY bRaised : BOOL
GET
bRaised := THIS^.fbTcAlarm.bRaised;
END_GET
END_PROPERTY

PROPERTY PUBLIC bSetEvent : BOOL
GET
bSetEvent := _bSetEvent;
END_GET
SET
_bSetEvent := bSetEvent;
END_SET
END_PROPERTY

METHOD Clear : HRESULT
VAR_INPUT
	nTimeStamp			: ULINT;
	bResetConfirmation	: BOOL;
END_VAR

IF NOT _bSetEvent AND_THEN THIS^.bActive THEN
	Clear := THIS^.fbTcAlarm.Clear( nTimeStamp, bResetConfirmation );
ELSE
	Clear := 1;
END_IF
END_METHOD

PROPERTY PUBLIC eEventReaction : E_AlarmReaction
GET
eEventReaction := _eEventReaction;
END_GET
SET // PUBLIC
_eEventReaction := eEventReaction;
END_SET
END_PROPERTY

PROPERTY eSeverity : TcEventSeverity
GET
eSeverity := THIS^.fbTcAlarm.eSeverity;
END_GET
END_PROPERTY

METHOD FB_exit : BOOL
VAR_INPUT
	bInCopyCode : BOOL;  // if TRUE, the instance afterwards gets moved into the copy code (online change)
END_VAR
VAR
	ipThis	: I_Alarm;
	ipPrev	: I_Alarm;
	nGuard	: UINT;
END_VAR
IF NOT bInCopyCode THEN
	THIS^.fbTcAlarm.ipArguments.Clear();
	THIS^.fbTcAlarm.Release();
	
	ipThis := THIS^;
	IF GVL_Diag.ipAlarmHead = ipThis THEN
		GVL_Diag.ipAlarmHead := _ipNext;
		IF GVL_Diag.gnCountAlarms > 0 THEN
			GVL_Diag.gnCountAlarms := GVL_Diag.gnCountAlarms - 1;
		END_IF
	ELSE
		ipPrev := GVL_Diag.ipAlarmHead;
		nGuard := 0;
		WHILE ipPrev <> 0 AND nGuard < Parameter.nMaxNumberAlarms DO
			nGuard := nGuard + 1;
			IF ipPrev.ipNext = ipThis THEN
				ipPrev.ipNext := _ipNext;
				IF GVL_Diag.gnCountAlarms > 0 THEN
					GVL_Diag.gnCountAlarms := GVL_Diag.gnCountAlarms - 1;
				END_IF
				EXIT;
			END_IF
			ipPrev := ipPrev.ipNext;
		END_WHILE
	END_IF
	_ipNext := 0;
END_IF
END_METHOD

METHOD FB_init : BOOL
VAR_INPUT
	bInitRetains : BOOL; // if TRUE, the retain variables are initialized (warm start / cold start)
	bInCopyCode : BOOL;  // if TRUE, the instance afterwards gets moved into the copy code (online change)
	
	stTmpEventClass	: TcEventEntry;
END_VAR

// no online-change
IF NOT bInCopyCode THEN
	
	// detect config error, if too many events were created during initializing
	IF GVL_Diag.gnCountAlarms >= Parameter.nMaxNumberAlarms THEN
		GVL_Diag.gbCountAlarmsMaxExceeded := TRUE;
	ELSE
		_stEventClass := stTmpEventClass;
		// standard event reaction depending of the event class severity
		CASE _stEventClass.eSeverity OF
			TcEventSeverity.Critical:
				_eEventReaction := E_AlarmReaction.MediaOff;
			TcEventSeverity.Error:
				_eEventReaction := E_AlarmReaction.AbortAll;
			TcEventSeverity.Warning:
				_eEventReaction := E_AlarmReaction.Warning;
			TcEventSeverity.Info:
				_eEventReaction := E_AlarmReaction.Info;
			TcEventSeverity.Verbose:
				_eEventReaction := E_AlarmReaction.Verbose;
		END_CASE
		
		{warning 'TODO: Understanding of Confirmation System'}
		// _bWithConfirmation := SEL( _stEventClass.eSeverity = TcEventSeverity.Error OR _stEventClass.eSeverity = TcEventSeverity.Critical, FALSE, TRUE);
		_bWithConfirmation := FALSE;
		
		THIS^.fbTcAlarm.CreateEx(
			_stEventClass,
			_bWithConfirmation,
			THIS^._fbInternalSourceInfo );
		
		Register();
		
	END_IF
	
END_IF
END_METHOD

METHOD PRIVATE Register : BOOL
VAR
	ipAlarm	: I_Alarm;
	ipThis	: I_Alarm;
	nGuard	: UINT;
END_VAR

ipThis := THIS^;

ipAlarm := GVL_Diag.ipAlarmHead;
nGuard := 0;
WHILE ipAlarm <> 0 AND nGuard < Parameter.nMaxNumberAlarms DO
	IF ipAlarm = ipThis THEN
		RETURN;
	END_IF
	ipAlarm := ipAlarm.ipNext;
	nGuard := nGuard + 1;
END_WHILE

IF GVL_Diag.gnCountAlarms >= Parameter.nMaxNumberAlarms THEN
	GVL_Diag.gbCountAlarmsMaxExceeded := TRUE;
	RETURN;
END_IF

_ipNext := GVL_Diag.ipAlarmHead;
GVL_Diag.ipAlarmHead := ipThis;
GVL_Diag.gnCountAlarms := GVL_Diag.gnCountAlarms + 1;
END_METHOD

METHOD GetEventEntry : ST_EventEntryTable
VAR_INPUT
END_VAR

GetEventEntry.sText := THIS^.sText;
GetEventEntry.sSourceName := THIS^.fbTcAlarm.ipSourceInfo.sName;
GetEventEntry.nSourceId := THIS^.fbTcAlarm.ipSourceInfo.nId;
GetEventEntry.nGroupId := THIS^.nGroupId;

GetEventEntry.sTimestamp := THIS^.sTimeRaised;

GetEventEntry.eSeverity := THIS^.fbTcAlarm.eSeverity;
CASE THIS^.fbTcAlarm.eSeverity OF
	TcEventSeverity.Verbose:	GetEventEntry.sSeverity := 'Verbose';
	TcEventSeverity.Info:		GetEventEntry.sSeverity := 'Info';
	TcEventSeverity.Warning:	GetEventEntry.sSeverity := 'Warning';
	TcEventSeverity.Error:		GetEventEntry.sSeverity := 'Error';
	TcEventSeverity.Critical:	GetEventEntry.sSeverity := 'Critical';
	ELSE	GetEventEntry.sSeverity := 'None';
END_CASE

CASE _eEventReaction OF
	E_AlarmReaction.AbortAll:	GetEventEntry.sReaction := 'Abort All';
	E_AlarmReaction.AbortGroup:	GetEventEntry.sReaction := 'Abort Group';
	E_AlarmReaction.Info:		GetEventEntry.sReaction := 'Info';
	E_AlarmReaction.MediaOff:	GetEventEntry.sReaction := 'Media Off';
	E_AlarmReaction.None:		GetEventEntry.sReaction := 'None';
	E_AlarmReaction.StopAtCycleEnd:	GetEventEntry.sReaction := 'StopAtCycleEnd';
	E_AlarmReaction.Verbose:	GetEventEntry.sReaction := 'Verbose';
	E_AlarmReaction.Warning:	GetEventEntry.sReaction := 'Warning';
	ELSE	GetEventEntry.sReaction := 'None';
END_CASE

GetEventEntry.EventClass := THIS^.fbTcAlarm.EventClass;
GetEventEntry.EventClassName := THIS^.sClassName;

GetEventEntry.nEventId := THIS^.fbTcAlarm.nEventId;
// GetEventEntry.ipArguments := fbTcAlarm.ipArguments;
GetEventEntry.eConfirmationState := THIS^.fbTcAlarm.eConfirmationState;
GetEventEntry.bIsAlarm := TRUE;
GetEventEntry.bIsEvent := FALSE;

GetEventEntry.nLanguageId := THIS^.nLangId;

(*
	sJsonAttribute: STRING(8000);
#	sText: STRING(255); // 
#	sSourceName: STRING(255); // 
#	nSourceId: UDINT; // 
	sDescription: STRING(255);
#	eSeverity: TcEventSeverity; // INT
#	sSeverity: STRING;
#	EventClass: GUID;
#	EventClassName: STRING(255); //
	sTimestampLog : STRING;
	sTimestamp: STRING; // 
	sTimestampConfirmed: STRING;
	sTimestampCleared: STRING;
#	nEventId: UDINT;
#	ipArguments: I_TcArguments;
#	eConfirmationState: TcEventConfirmationState; // 
	bTextReceived: BOOL;
#	bIsAlarm: BOOL;
#	bIsEvent: BOOL;
	stAlarmLog : ST_AlarmLog;
	bLogged : BOOL;
#	nLanguageId : INT;
*)
END_METHOD

METHOD GetEventText : BOOL
VAR_INPUT
END_VAR
VAR_INST
	bReqTextError	: BOOL;
END_VAR

GetEventText := FALSE;

IF THIS^.fbTcAlarm.RequestEventText(
	nLangId		:= 1031,
	sResult		:= sText,
	nResultSize	:= SIZEOF( sText ),
	bError		=> bReqTextError
) THEN
	GetEventText := TRUE;
END_IF

IF bReqTextError THEN
	sText := '';
END_IF
END_METHOD

METHOD GetJsonAttribute : HRESULT
VAR_INPUT
	sJsonAttribute	: REFERENCE TO STRING;
	nJsonAttribute	: UDINT;
END_VAR

THIS^.fbTcAlarm.GetJsonAttribute( sJsonAttribute, nJsonAttribute );
END_METHOD

METHOD PUBLIC Initialize : HRESULT
VAR_INPUT
	nTmpZoneId			: UINT;
	nTmpGroupId			: UINT;
	eInEventReaction	: E_AlarmReaction;
END_VAR

THIS^.nZoneId := nTmpZoneId;
THIS^.nGroupId := nTmpGroupId;
THIS^._eEventReaction := eInEventReaction;
Register();
END_METHOD

PROPERTY PUBLIC ipArguments : I_TcArguments
GET
ipArguments := THIS^.fbTcAlarm.ipArguments;
END_GET
END_PROPERTY

PROPERTY ipNext : I_Alarm
GET
ipNext := _ipNext;
END_GET
SET
_ipNext := ipNext;
END_SET
END_PROPERTY

PROPERTY PUBLIC LogEntry : ST_LogEntry
GET

LogEntry.sText := sText;
LogEntry.sTimestampLog := sTimeRaised;
LogEntry.sSeverity := THIS^.sSeverity;
LogEntry.sSourceName := THIS^._fbInternalSourceInfo.sName;
END_GET
END_PROPERTY

PROPERTY PUBLIC nGetGroupId : UINT
GET
nGetGroupId := nGroupId;
END_GET
END_PROPERTY

PROPERTY PUBLIC nGetSourceId : UDINT
GET
nGetSourceId := THIS^.fbTcAlarm.ipSourceInfo.nId;
END_GET
END_PROPERTY

METHOD Raise : HRESULT
VAR_INPUT
	nTimeStamp	: ULINT;
END_VAR
THIS^.fbTcAlarm.Raise( 0 );

THIS^.sTimeRaised := SYSTEMTIME_TO_STRING(
	UlintToSystemTime(
		THIS^.fbTcAlarm.nTimeRaised,
		GVL_Diag.gfbAlarmManagement.fbGetTimeZoneInformation.tzInfo ) );
END_METHOD

METHOD PUBLIC SetEvent : REFERENCE TO FB_Alarm
VAR_INPUT
	bSetEvent	: BOOL;
END_VAR

IF bSetEvent
AND_THEN NOT THIS^._bSetEvent
AND_THEN NOT THIS^.bActive THEN
	hrRaise := THIS^.Raise( 0 );
	GVL_Diag.gfbLogFile.addEntry( THIS^ );
END_IF
_bSetEvent := bSetEvent;
_bBlockAck S= bSetEvent;

setEvent REF= THIS^;
END_METHOD

METHOD PUBLIC SetEventWithOneArgument : REFERENCE TO FB_Alarm
VAR_INPUT
	bSetEvent		: BOOL;
	sInName			: STRING;
END_VAR
VAR_INST
	rtSetEvent		: R_TRIG;
END_VAR
VAR
    hr		: HRESULT;
    UTF8	: STRING(255);
END_VAR

IF bSetEvent
AND_THEN NOT THIS^._bSetEvent
AND_THEN NOT THIS^.bActive THEN
	THIS^.start().addArgument( sInName );
	hrRaise := THIS^.Raise( 0 );
	GVL_Diag.gfbLogFile.addEntry( THIS^ );
END_IF
_bSetEvent := bSetEvent;
_bBlockAck S= _bSetEvent;

setEventWithOneArgument REF= THIS^;
END_METHOD

PROPERTY PRIVATE sSeverity : STRING
GET

CASE fbTcAlarm.eSeverity OF
	
	TcEventSeverity.Critical:
		sSeverity := 'Critical';
		
	TcEventSeverity.Error:
		sSeverity := 'Error';
		
	TcEventSeverity.Info:
		sSeverity := 'Info';
		
	TcEventSeverity.Verbose:
		sSeverity := 'Verbose';
		
	TcEventSeverity.Warning:
		sSeverity := 'Warning';
		
	ELSE
		sSeverity := 'None';
		
END_CASE
END_GET
END_PROPERTY

METHOD PUBLIC Start : REFERENCE TO FB_Alarm
VAR_INPUT
END_VAR

THIS^.fbTcAlarm.ipArguments.Clear();
start REF= THIS^;
_nArgumentCount := 0;
END_METHOD

METHOD PRIVATE UlintToSystemTime : TIMESTRUCT
VAR_INPUT
	_fileTime: ULINT;
	_tzInfo: ST_TimeZoneInformation;
END_VAR
VAR
	tfileTime: T_FILETIME;
	tfileTimeZone: T_FILETIME;
	fbFileTimeToTzSpecificLocalTime: FB_FileTimeToTzSpecificLocalTime;
END_VAR

MEMCPY( ADR( tfileTime ),ADR( _fileTime ), SIZEOF( T_FILETIME ) );
fbFileTimeToTzSpecificLocalTime(
	in := tfileTime, 
	tzInfo := _tzInfo, 
	out => tfileTimeZone, 
	eTzID => , 
	bB => );
UlintToSystemTime := FILETIME_TO_SYSTEMTIME( fileTime:= tfileTimeZone );
END_METHOD

METHOD PUBLIC UpdateText : HRESULT
VAR_INPUT
	LangId	: INT;
END_VAR
VAR_INST
    nStep : E_AlarmMessage;
    nStepRequestText : E_AlarmMessage := E_AlarmMessage.Done;
    nStepRequestClass : E_AlarmMessage := E_AlarmMessage.Done;
END_VAR
VAR
	
    hr : HRESULT;
    UTF8 : STRING(255);
END_VAR

IF ( nStepRequestText <> E_AlarmMessage.Done
	OR nStepRequestClass <> E_AlarmMessage.Done )
AND THIS^.bRaised THEN
	
	// CASE: RequestText   
	IF nStepRequestText = E_AlarmMessage.RequestText THEN
		THIS^.fbRequestText.Request( eventClass := THIS^.fbTcAlarm.EventClass, nEventId := THIS^.fbTcAlarm.nEventId, nLangId := LangId, ipArgs := THIS^.fbTcAlarm.ipArguments );
		nStepRequestText := E_AlarmMessage.ReceiveText;
	END_IF
	
	// CASE: ReceiveText   
	IF nStepRequestText = E_AlarmMessage.ReceiveText THEN
		IF NOT THIS^.fbRequestText.bBusy AND NOT THIS^.fbRequestText.bError THEN
			THIS^.fbRequestText.GetString( UTF8, SIZEOF( UTF8 ) );
			UTF8_TO_STRING(pDstSTRING := ADR( sText ), pSrcUTF8 := ADR( UTF8 ), nDstSize := SIZEOF( sText ), nDstLen => );
			nStepRequestText := E_AlarmMessage.Done;
		ELSIF THIS^.fbRequestText.bError THEN 
			nStepRequestText := E_AlarmMessage.RequestText;
		END_IF
	END_IF
	
    // CASE: RequestClassText   
    IF nStepRequestClass = E_AlarmMessage.RequestText THEN
		THIS^.fbRequestClassName.Request( eventClass := THIS^.fbTcAlarm.EventClass, nLangId := LangId );
		nStepRequestClass := E_AlarmMessage.ReceiveText;
	END_IF
	
    // CASE: ReceiveClassText   
    IF nStepRequestClass = E_AlarmMessage.ReceiveText THEN
        IF NOT THIS^.fbRequestClassName.bBusy AND NOT THIS^.fbRequestClassName.bError THEN
            THIS^.fbRequestClassName.GetString( UTF8, SIZEOF( UTF8 ) );
            UTF8_TO_STRING(pDstSTRING:=ADR( sClassName ), pSrcUTF8 := ADR( UTF8 ), nDstSize:=SIZEOF( sClassName ), nDstLen=> );
            nStepRequestClass := E_AlarmMessage.Done;
        ELSIF THIS^.fbRequestClassName.bError THEN 
            nStepRequestClass := E_AlarmMessage.RequestText;
        END_IF
	END_IF

ELSE
	// reset Text
	IF NOT bRaised OR nLangId <> LangId THEN
		sText := '';
		sClassName := '';
		nStepRequestClass := E_AlarmMessage.RequestText;
		nStepRequestText := E_AlarmMessage.RequestText;
		nLangId := LangId;
	END_IF
END_IF

IF THIS^.fbRequestClassName.bError
OR THIS^.fbRequestText.bError THEN
	UpdateText := E_FAIL;
ELSIF THIS^.fbRequestClassName.bBusy
OR THIS^.fbRequestText.bBusy THEN
	UpdateText := S_OK;
ELSE
	UpdateText := S_PENDING;
END_IF
END_METHOD

END_FUNCTION_BLOCK

// ---- EventLogger/Logger/FB_LogFile.TcPOU
FUNCTION_BLOCK FB_LogFile
VAR_INPUT
END_VAR
VAR_OUTPUT
END_VAR
VAR
	aiLogEntry	: ARRAY[0..MAX_INDEX] OF I_Message;
	astLogEntry	: ARRAY[0..MAX_INDEX] OF ST_LogEntry;
	indexNew	: UINT := 0;
	index		: UINT := 0;
	
	stLogEntry	: ST_LogEntry;
	
    _logCache   : FB_LogStringBuffer; // Dynamic string buffer to cache logs to be processed
    fbFileRetentionTimeHandler : FB_FileRetentionTimeHandler;
    _bOverflow	: BOOL;
    DebugString	: STRING( Parameter.MAX_LOG_STRING_SIZE );
    lastLogTimeAsStruct	: TIMESTRUCT;
    fbFileOpen  : FB_FileOpen;
    fbFileWrite : FB_FileWrite;
	
	fbState		: FB_StateMachine;
	
	// config
    _fileName	: T_MaxString := '';
    _CfgFileName	: T_MaxString := 'log'; // Base file name
    _filePath	: T_MaxString := 'C:\Logs\'; // Path to folder 
    _RollingInterval	: E_RollingInterval := E_RollingInterval.Daily; // Interval when to start a new file
	_delimiter	: STRING( 3 ) := ' | ';
    _LogFileLifespan	: UINT := 30; // Lifespan of logfiles in days. Once exceeded, log files will be deleted.
    _TimestampFormat	: STRING := 'YYYYMMDD_hhmm'; // Format the timestamp should have
	
	// time and date
    _TimeData	: FB_GenerateTimeData;
    timeAsFileTime   : T_FILETIME; // Actual time as filetime, corrected to local time zone
    lastTimeCallTime : LINT;
    timeAsSystemTime : TIMESTRUCT; // Actual time as timestring
    timeAsString : STRING; // Actual time as string
	
    _timeStamp : STRING( 255 );
	
    bInit	: BOOL;
END_VAR
VAR CONSTANT
	MAX_INDEX	: UINT := 9999;
END_VAR

GetTime();

// run logger
IF NOT bInit THEN
	fbFileRetentionTimeHandler.Configure( _LogFileLifespan, _filePath, _fileName, _TimeData );
	bInit := TRUE;
END_IF

// Generate new timestamp for filename
IF RollingIntervalReached( lastlogTimeAsStruct, _RollingInterval ) OR _TimeData.Done THEN
	_timeStamp := _TimeData.ToString( _TimestampFormat );
	_filePath := SEL( RIGHT( _filePath, 1 ) <> '\', _filePath, CONCAT( _filePath, '\' ) );
	
	fbConcat.SetDstString( _fileName )
		.AddString( _filePath )
		.AddString( _timeStamp )
		.AddStringInput( '.' )
		.AddString( _CfgFileName ).Get();

END_IF

// Delete expired log files
fbFileRetentionTimeHandler.HandleFiles();

IF _TimeData.IsValid AND _filename <> '' THEN
	// Persist logging messages to file
	PersistToFile( _filename );
END_IF

// automatic detection of new entries
CASE fbState.nState OF

	0:	// wait for new entries
		IF index <> indexNew THEN
			fbState.IncrementState( 1 );
		END_IF
	
	1:	// check entry, trigger eventlogger if necessary
		stLogEntry.sText := '';
		
		// log entry from TC EventClass
		IF aiLogEntry[index] <> 0 THEN
			IF aiLogEntry[index].GetEventText() THEN
				stLogEntry := aiLogEntry[index].LogEntry;
			END_IF
			
		// log from structure
		ELSIF astLogEntry[index].sText <> '' THEN
			stLogEntry := astLogEntry[index];
		END_IF
		
		// text available, next step
		IF stLogEntry.sText <> '' THEN
			LogData(
				Message := stLogEntry.sText,
				Source := stLogEntry.sSourceName,
				Severity := stLogEntry.sSeverity,
				timeAsString := stLogEntry.sTimestampLog
			);
			IF index < MAX_INDEX THEN
				index := index + 1;
			ELSE
				index := 0;
			END_IF
			
			fbState.IncrementState( 1 );
		END_IF
	
	2:	// wait log data done
		fbState.SetNextState( 0 );
		
END_CASE

METHOD addEntry : BOOL
VAR_INPUT
	entry	: I_Message;
END_VAR
VAR
	i	: INT;
END_VAR

addEntry := TRUE;

// add entry interface at current index, no shifting of array.
aiLogEntry[indexNew] := entry;

IF indexNew >= MAX_INDEX
AND_THEN index <> 0 THEN
	indexNew := 0;
ELSIF ( indexNew + 1 ) <> index THEN
	indexNew := indexNew + 1;
END_IF
END_METHOD

METHOD addLog : BOOL
VAR_INPUT
	entry	: STRING;
END_VAR
VAR
	i	: INT;
END_VAR

addLog := TRUE;

{warning 'TODO: timestamp withing Logger, also convenient way to get source info and severity'}
astLogEntry[indexNew].sText := entry;
astLogEntry[indexNew].sSeverity := 'manually';

IF indexNew >= MAX_INDEX
AND_THEN index <> 0 THEN
	indexNew := 0;
ELSIF ( indexNew + 1 ) <> index THEN
	indexNew := indexNew + 1;
END_IF
END_METHOD

{attribute 'hide'}
METHOD GetTime : BOOL
VAR_INPUT
END_VAR
VAR
    nTaskIdx            : DINT;
    currentTimeCallTime : LINT;
END_VAR

nTaskIdx := GETCURTASKINDEXEX();

IF nTaskIdx > 0 THEN
	currentTimeCallTime := TwinCAT_SystemInfoVarList._TaskInfo[nTaskIdx].DcTaskTime;
	
	IF lastTimeCallTime = currentTimeCallTime THEN
		RETURN; // Only call once per cycle
	END_IF
	
	// Generate time data (shared state)
	fbSystemTime();
	_TimeData(
		timeAsFileTime => timeAsFileTime,
		timeAsSystemTime => timeAsSystemTime,
		timeAsString => timeAsString
	);
	lastTimeCallTime := currentTimeCallTime;
END_IF
END_METHOD

{attribute 'hide'}
METHOD LogData : BOOL
VAR_IN_OUT CONSTANT
    Message			: STRING( Parameter.MAX_LOG_STRING_SIZE ); // Message to log.
    Source			: T_MaxString;	// source info of logEntry
    Severity		: STRING;
    timeAsString	: STRING;		// timestamp as string
END_VAR
VAR
END_VAR

IF _bOverflow AND _logCache.IsEmpty THEN
    _bOverflow := FALSE;
END_IF

IF NOT _bOverflow THEN

    IF _fileName <> '' THEN
        fbConcat.SetDstString( DebugString )
            .AddStringInput( timeAsString )
            .AddString( _delimiter )
            .AddStringInput( Severity )
            .AddString( _delimiter )
            .AddStringInput( Source )
            .AddString( _delimiter )
            .AddStringInput( Message );

        IF NOT _LogCache.AddLine( DebugString ) THEN
            _bOverflow := TRUE;
        END_IF
		
    END_IF
	
END_IF
END_METHOD

{attribute 'hide'}
METHOD PersistToFile : BOOL
VAR_INPUT
    FileName : T_MAXSTRING; //	File name including its path
END_VAR
VAR_INST
    state : UINT;

    fbFileOpen      : FB_FileOpen;
    fTrigFileOpened : F_TRIG;
    hFile           : UINT;

    fbFilePuts        : FB_FileWrite;
    fTrigFilePuts     : F_TRIG;
    newLogEntry       : STRING( Parameter.MAX_LOG_STRING_SIZE * Parameter.MAX_BUFFER_COUNT );
    filePutsTriggered : BOOL;

    fbFileClose    : FB_FileClose;
    fTrigFileClose : F_TRIG;
    tonTimeout     : TON;
    bDebug         : BOOL;
END_VAR
VAR CONSTANT
    STATE_IDLE                 : UINT := 0;
    STATE_OPEN_FILE            : UINT := 1;
    STATE_GET_STRING_FROM_FIFO : UINT := 2;
    STATE_APPEND_DATA_TO_FILE  : UINT := 3;
    STATE_CLOSE_FILE           : UINT := 4;

    NET_ID  : STRING := '';
    TIMEOUT : TIME := T#20S;
END_VAR

// State machine
CASE state OF
	STATE_IDLE:
		IF NOT _logCache.IsEmpty THEN
			filePutsTriggered := FALSE;
			state := STATE_OPEN_FILE;
		END_IF
	
	STATE_OPEN_FILE:
		IF fTrigFileOpened.Q THEN
			state := STATE_GET_STRING_FROM_FIFO;
		END_IF
	
	STATE_GET_STRING_FROM_FIFO:
		MEMSET( ADR( newLogEntry ), 0, SIZEOF( newLogEntry ) );
	
		IF NOT filePutsTriggered THEN
			_logCache.PopHead( resultString := newLogEntry );
			state := STATE_APPEND_DATA_TO_FILE;
		END_IF
	
		filePutsTriggered := FALSE;
	
	STATE_APPEND_DATA_TO_FILE:
		filePutsTriggered := TRUE;
	
		IF fTrigFilePuts.Q THEN
			IF NOT _logCache.IsEmpty AND NOT tonTimeout.Q THEN
				state := STATE_GET_STRING_FROM_FIFO;
			ELSE
				state := STATE_CLOSE_FILE;
			END_IF
		END_IF
	
	STATE_CLOSE_FILE:
		IF fTrigFileClose.Q THEN
			state := STATE_IDLE;
		END_IF

END_CASE

// Function blocks used in state machine
fbFileOpen(
	sNetId := NET_ID,
	sPathName := FileName,
	nMode := FOPEN_MODEAPPEND OR FOPEN_MODETEXT,
	ePath := PATH_GENERIC,
	bExecute := ( state = STATE_OPEN_FILE ),
	tTimeout := TIMEOUT,
	hFile => hFile
);

fTrigFileOpened( CLK := fbFileOpen.bBusy );

fbFilePuts(
	sNetId := NET_ID,
	hFile := hFile,
	pWriteBuff := ADR( newLogEntry ),
	cbWriteLen := LEN2( ADR( newLogEntry ) ),
	bExecute := ( state = STATE_APPEND_DATA_TO_FILE ),
	tTimeout := TIMEOUT
);

fTrigFilePuts( CLK := fbFilePuts.bBusy );

fbFileClose(
	sNetId := NET_ID,
	hFile := hFile,
	bExecute := ( state = STATE_CLOSE_FILE ),
	tTimeout := TIMEOUT
);

fTrigFileClose( CLK := fbFileClose.bBusy );

//IF tonTimeout.Q AND NOT bDebug THEN
//    state := STATE_IDLE;
//END_IF
// Timeout writing to file => close file
tonTimeout( IN := state <> STATE_IDLE, PT := TIMEOUT );

// Error handling
//IF fbFileOpen.bError THEN
//    Error.Active := TRUE;
//    Error.Code := E_ErrorCode.OpeningFileFailed;
//    Error.Info := CONCAT('Opening file failed. Error thrown by FB_FileOpen. Consult Beckhoff InfoSys. Internal Error: ', UDINT_TO_STRING(fbFileOpen.nErrId));
//ELSIF fbFilePuts.bError THEN
//    Error.Active := TRUE;
//    Error.Code := E_ErrorCode.WritingToFileFailed;
//    Error.Info :=
//        CONCAT('Writing to file failed. Error thrown by FB_FilePuts. Consult Beckhoff InfoSys. Internal Error: ', UDINT_TO_STRING(fbFilePuts.nErrId));
//ELSIF fbFileClose.bError THEN
//    Error.Active := TRUE;
//    Error.Code := E_ErrorCode.ClosingFileFailed;
//    Error.Info := CONCAT('Closing file failed. Error thrown by FB_FileClose. Consult Beckhoff InfoSys. Internal Error: ', UDINT_TO_STRING(fbFileClose.nErrId));
//ELSIF NOT Fifo.bOk AND Fifo.nCount > 0 THEN
//    Error.Active := TRUE;
//    Error.Code := E_ErrorCode.FifoOverflow;
//    Error.Info := 'FIFO overflow. Check if (a) plc has enough free memory and (b) if no message is written each plc cycle';
//ELSE
//    Error.Active := FALSE;
//    Error.Code := E_ErrorCode.None;
//    Error.Info := '';
//END_IF
END_METHOD

// Checks the specified rolling interval for the file name.
// Generates new file name if rolling intervall exceeded.
{attribute 'hide'}
METHOD PRIVATE RollingIntervalReached : BOOL
VAR_INPUT
    actualTime      : TIMESTRUCT;
    rollingInterval : E_RollingInterval;
END_VAR
VAR_INST
    lastTime : TIMESTRUCT;
END_VAR

IF actualTime.wYear > lastTime.wYear OR actualTime.wMonth > lastTime.wMonth THEN
    // new year or month is also new hour and new day
    RollingIntervalReached := TRUE;
ELSIF actualTime.wDay > lastTime.wDay THEN
    // new day is also new hour
    RollingIntervalReached := rollingInterval = E_RollingInterval.Hourly OR rollingInterval = E_RollingInterval.Daily;
ELSIF actualTime.wHour > lastTime.wHour THEN
    // new hour only holds for hourly
    RollingIntervalReached := rollingInterval = E_RollingInterval.Hourly;
END_IF

// save actual log time as last time
MEMCPY( ADR( lastTime ), ADR( actualTime ), SIZEOF( actualTime ) );
END_METHOD

END_FUNCTION_BLOCK

// ---- EventLogger/Logger/FB_LogStringBuffer.TcPOU
FUNCTION_BLOCK FB_LogStringBuffer
VAR_INPUT
END_VAR
VAR_OUTPUT
END_VAR
VAR
    fbFifoBuffer : FB_MemRingBuffer; // Necessary to buffer log data until it has been written to file.
    asBuffer     : ARRAY[0..STRING_BUFFER_SIZE] OF BYTE; // Buffer of string
    headString   : STRING( Parameter.MAX_LOG_STRING_SIZE + 1 );
    nHeadLen     : UDINT;
    ConcatText   : STRING( Parameter.MAX_LOG_STRING_SIZE + 1 );
    newline      : STRING( 1 ) := '$N';
END_VAR
VAR CONSTANT
    BUFFER_OVERHEAD    : UDINT := 10;
    STRING_BUFFER_SIZE : UDINT := ( Parameter.MAX_LOG_STRING_SIZE + BUFFER_OVERHEAD ) * Parameter.MAX_BUFFER_COUNT;
END_VAR

METHOD AddLine : BOOL
VAR_IN_OUT 
    Text : STRING( Parameter.MAX_LOG_STRING_SIZE );
END_VAR
VAR
    pText : POINTER TO BYTE;
END_VAR

pText := ADR( Text );
CONCAT2( pText, ADR( newline ), ADR( ConcatText ), SIZEOF( ConcatText ) );

fbFifoBuffer.A_AddTail(
	pWrite := ADR( ConcatText ),
	cbWrite := LEN2( ADR( ConcatText ) )
);

AddLine := fbFifoBuffer.bOk;
END_METHOD

METHOD AddString : BOOL
VAR_INPUT
    Text : STRING( Parameter.MAX_LOG_STRING_SIZE );
END_VAR

fbFifoBuffer.A_AddTail(
	pWrite := ADR( Text ),
	cbWrite := LEN2( ADR( Text ) )
);
AddString := fbFifoBuffer.bOk;
END_METHOD

METHOD PRIVATE AllocateBuffer : BOOL
VAR_INPUT
END_VAR

fbFifoBuffer.pBuffer := ADR( asBuffer );
fbFifoBuffer.cbBuffer := SIZEOF( asBuffer );
END_METHOD

METHOD FB_init : BOOL
VAR_INPUT
	bInitRetains : BOOL; // if TRUE, the retain variables are initialized (warm start / cold start)
	bInCopyCode : BOOL;  // if TRUE, the instance afterwards gets moved into the copy code (online change)
END_VAR
AllocateBuffer();
END_METHOD

METHOD FB_reinit : BOOL
VAR_INPUT
END_VAR
AllocateBuffer();
END_METHOD

METHOD FlushCache : BOOL
VAR_INPUT
END_VAR
fbFifoBuffer.A_Reset();
END_METHOD

PROPERTY IsEmpty : BOOL
GET
IsEmpty := fbFifoBuffer.nCount = 0;
END_GET
END_PROPERTY

METHOD PopHead : BOOL
VAR_IN_OUT
    resultString : STRING( Parameter.MAX_LOG_STRING_SIZE * 2 );
END_VAR
VAR
    pResult        : POINTER TO BYTE;
    nRemainingSize : UDINT;
    pHead          : POINTER TO BYTE;
    nHeadSize      : UDINT;
    nFifoCount     : UDINT;
END_VAR

// create pointer and size for result
pResult := ADR( resultString );
nRemainingSize := SIZEOF( resultString );

// Clear result
MEMSET( pResult, 0, nRemainingSize );

// Check current buffered strings
nFifoCount := fbFifoBuffer.nCount;

IF nFifoCount = 0 THEN
    RETURN;
END_IF

// Create pointer and size for head string
pHead := ADR( headString );
nHeadSize := SIZEOF( headString );

REPEAT
    // Clear head data
    MEMSET( pHead, 0, nHeadSize );
    // get (not pop) head data
    fbFifoBuffer.A_GetHead( pRead := pHead, cbRead := nHeadSize );
    // get string size
    nHeadLen := LEN2( pHead );

    // Check if head still fits into result string
    IF nRemainingSize - nHeadLen - 1 > 0 THEN
        // If it fits 
        PopHead := TRUE;

        // Copy data
        MEMCPY( pResult, pHead, nHeadLen );

        // Move pointer to next result position and set remaining size
        pResult := pResult + nHeadLen;
        nRemainingSize := nRemainingSize - nHeadLen;

        // Remove the copied entry
        fbFifoBuffer.A_RemoveHead();
        nFifoCount := nFifoCount - 1;
    END_IF
UNTIL

	// unless it does not fit any more or no further buffered data
    nRemainingSize - nHeadLen - 1 <= 0 OR nFifoCount = 0
END_REPEAT;
END_METHOD

END_FUNCTION_BLOCK

// ---- EventLogger/Logger/FB_FileRetentionTimeHandler.TcPOU
FUNCTION_BLOCK FB_FileRetentionTimeHandler
VAR_INPUT
END_VAR
VAR_OUTPUT
END_VAR
VAR
    _expirationInDays : UINT; // 	Files will be deleted if older than n days
    _filePath         : T_MAXSTRING; //	Path to files to be deleted
    _fileName         : T_MAXSTRING; //	Only files which match this filename will be deleted
    _timeProvider     : REFERENCE TO FB_GenerateTimeData;
    _actualTime       : T_FILETIME; // 	Actual Time
    _actualSysTime    : TIMESTRUCT;

    fbEnum              : FB_EnumFindFileList;
    bRunSearch          : BOOL;
    fbDeleteFile        : FB_FileDelete;
    fTrigDeleteFileBusy : F_TRIG;
    _state              : UINT := 0;
    filesList           : ARRAY[0..MAX_FILES_COUNT - 1] OF ST_FindFileEntry;
    deleteFileIndex     : UDINT;
    deleteFileName      : T_MAXSTRING;
    eEnumCmd            : E_EnumCmdType;
    _LastDay            : TIMESTRUCT;
    _sSearchPath        : T_MaxString;
    bRemoveFile         : BOOL;
END_VAR
VAR CONSTANT
    GetFilesState      : UINT := 0;
    RemoveFilesState   : UINT := 1;
    MAX_FILES_COUNT    : INT := 100;
    ONE_DAY_IN_SECONDS : LREAL := 24 * 3600.0;
END_VAR

METHOD Configure : BOOL
VAR_INPUT
    expirationInDays : UINT; // 	Files will be deleted if older than n days
    filePath         : T_MAXSTRING; //	Path to files to be deleted
    fileName         : T_MAXSTRING; //	Only files which match this filename will be deleted
    timeProvider     : REFERENCE TO FB_GenerateTimeData;
END_VAR

_expirationInDays := expirationInDays;
_filePath := filePath;
_fileName := fileName;
_timeProvider REF= timeProvider;
END_METHOD

METHOD HandleFiles : BOOL
VAR_INPUT
END_VAR

IF NOT _timeProvider.IsValid THEN
    // We cannot work without valid time data
    RETURN;
END_IF

_timeProvider( timeAsSystemTime => _actualSysTime, timeAsFileTime => _actualTime );

IF _LastDay.wDay = _actualSysTime.wDay
AND _LastDay.wMonth = _actualSysTime.wMonth
AND _LastDay.wYear = _actualSysTime.wYear THEN
    // Still same day, nothing to do
    RETURN;
END_IF

CASE _state OF
	GetFilesState:
		HandleFileSearch();
	RemoveFilesState:
		HandleRemoveCommands();
END_CASE

// Search files in given directory
fbEnum(
	sNetId := '',
	eCmd := eEnumCmd,
	sPathName := _sSearchPath,
	bExecute := bRunSearch,
	pFindList := ADR( filesList ),
	cbFindList := SIZEOF( filesList ),
	tTimeout := T#10S
);

// Delete files
fbDeleteFile( sNetId := '', sPathName := deleteFileName, bExecute := bRemoveFile, tTimeout := T#10S );
END_METHOD

METHOD PRIVATE HandleFileSearch : BOOL
VAR_INPUT
END_VAR
bRemoveFile := FALSE;
eEnumCmd := eEnumCmd_First;
deleteFileIndex := 0;
_sSearchPath := CONCAT(_filePath, CONCAT('*', _fileName));

IF bRunSearch AND NOT fbEnum.bBusy AND NOT fbEnum.bError AND fbEnum.nFindFiles > 0 THEN
    // end search and remove files
    // set abort command if EoE reached otherwise not necessary
    eEnumCmd := SEL(fbEnum.bEOE, eEnumCmd_Abort, eEnumCmd_First);
    _state := RemoveFilesState;
ELSIF bRunSearch AND NOT fbEnum.bBusy AND fbEnum.nFindFiles = 0 THEN
    // Nothing has been found, wait for next day
    _LastDay := _actualSysTime;
    bRunSearch := FALSE;
ELSIF bRunSearch AND fbEnum.bError THEN
    // if error restart search
    bRunSearch := FALSE;
ELSE
    // start search
    bRunSearch := TRUE;
END_IF
END_METHOD

METHOD PRIVATE HandleRemoveCommands : BOOL
VAR_INPUT
END_VAR
END_METHOD

END_FUNCTION_BLOCK

// ---- EventLogger/Logger/FB_GenerateTimeData.TcPOU
FUNCTION_BLOCK FB_GenerateTimeData
VAR_INPUT
END_VAR
VAR_OUTPUT
    timeAsFileTime    : T_FILETIME;
    timeAsSystemTime  : TIMESTRUCT;
    dateTimeAsString  : T_MaxString;
    timeAsString      : T_MaxString;
    utcTimeAsFileTime : T_FILETIME;
END_VAR
VAR
    fbTimeZoneInfo : FB_GetTimeZoneInformation;
    rTrigTimeValid : R_TRIG;
    fbUTCTime      : FB_TzSpecificLocalTimeToFileTime;
END_VAR


timeAsSystemTime := fbSystemTime.TimeStruct;

fbTimeZoneInfo( sNetID := '', bExecute := TRUE, tTimeout := DEFAULT_ADS_TIMEOUT );

fbUTCTime(in := SYSTEMTIME_TO_FILETIME( timeAsSystemTime ), tzInfo := fbTimeZoneInfo.tzInfo );

timeAsFileTime := SYSTEMTIME_TO_FILETIME( fbSystemTime.TimeStruct );
dateTimeAsString := fbSystemTime.ToString;

DELETE2(
	pSrcString := ADR( dateTimeAsString ),
	pDstString := ADR( timeAsString ),
	nDstSize := SIZEOF( timeAsString ),
	nLen := 11,
	nPos := 1
);

utcTimeAsFileTime := fbUTCTime.out;

rTrigTimeValid( CLK := fbSystemTime.IsValid );

PROPERTY Done : BOOL
GET
Done := rTrigTimeValid.Q;
END_GET
END_PROPERTY

PROPERTY IsValid : BOOL
GET
IsValid := fbSystemTime.IsValid;
END_GET
END_PROPERTY

METHOD PRIVATE ReplaceFormatPlaceHolder : STRING
VAR_INPUT
    Format   : STRING;
    Length   : INT;
    TimeType : STRING(1);
END_VAR
VAR
    i             : INT;
    replaceString : STRING;
    timeString    : STRING;
END_VAR

IF TimeType = 'Y' THEN
    timeString := TO_STRING( timeAsSystemTime.wYear );
ELSIF TimeType = 'M' THEN
    timeString := TO_STRING( timeAsSystemTime.wMonth );
ELSIF TimeType = 'D' THEN
    timeString := TO_STRING( timeAsSystemTime.wDay );
ELSIF TimeType = 'h' THEN
    timeString := TO_STRING( timeAsSystemTime.wHour );
ELSIF TimeType = 'm' THEN
    timeString := TO_STRING( timeAsSystemTime.wMinute );
ELSIF TimeType = 's' THEN
    timeString := TO_STRING( timeAsSystemTime.wSecond );
ELSIF TimeType = 'i' THEN
    timeString := TO_STRING( timeAsSystemTime.wMilliseconds );
END_IF

replaceString := '';

IF Length > LEN( timeString ) THEN
    FOR i := 1 TO Length - LEN( timeString ) DO
        replaceString := CONCAT( replaceString, '0' );
    END_FOR

    replaceString := CONCAT( replaceString, timeString );
ELSE
    replaceString := RIGHT( timeString, Length );
END_IF

ReplaceFormatPlaceholder := REPLACE( Format, replaceString, Length, FIND( Format, TimeType ) );
END_METHOD

(*
| Returns a formatted string containing the actual time information
|   `Y : year`
|   `M : month`
|   `D : day`
|   `h : hour` 
|   `m : minute`
|   `s : second`
|   `i : millisecond`

Example: `_YYMMDD-hh:mm:ss:iii_` => `_20210812-12:30:22:123_`
*)
METHOD ToString : T_MAXSTRING
VAR_INPUT
    Format : STRING;
END_VAR
VAR
    inputString     : STRING;
    sChar            : STRING(1);
    formattedString : T_MAXSTRING;

    year        : INT := 0;
    month       : INT := 0;
    day         : INT := 0;
    hour        : INT := 0;
    minute      : INT := 0;
    second      : INT := 0;
    millisecond : INT := 0;
END_VAR
VAR CONSTANT
    VALID_FORMAT : STRING := 'YMDhms';
END_VAR

// Parses "Format" and returns a adequatly formatted string containing the time information

inputString := Format;

WHILE LEN(inputString) > 0 DO
    sChar := LEFT(inputString, 1);

    IF sChar = 'Y' THEN
        year := year + 1;
    ELSIF sChar = 'M' THEN
        month := month + 1;
    ELSIF sChar = 'D' THEN
        day := day + 1;
    ELSIF sChar = 'h' THEN
        hour := hour + 1;
    ELSIF sChar = 'm' THEN
        minute := minute + 1;
    ELSIF sChar = 's' THEN
        second := second + 1;
    ELSIF sChar = 'i' THEN
        millisecond := millisecond + 1;
    END_IF

    inputString := DELETE( inputString, 1, 1 );
END_WHILE

formattedString := ReplaceFormatPlaceholder( Format, year, 'Y' );
formattedString := ReplaceFormatPlaceholder( formattedString, month, 'M' );
formattedString := ReplaceFormatPlaceholder( formattedString, day, 'D' );
formattedString := ReplaceFormatPlaceholder( formattedString, hour, 'h' );
formattedString := ReplaceFormatPlaceholder( formattedString, minute, 'm' );
formattedString := ReplaceFormatPlaceholder( formattedString, second, 's' );
formattedString := ReplaceFormatPlaceholder( formattedString, millisecond, 'i' );

ToString := formattedString;
END_METHOD

END_FUNCTION_BLOCK

// ---- StateMachine/FB_StateMachine.TcPOU
FUNCTION_BLOCK FB_StateMachine
(* Sequencer: in CASE nState add conditions each cycle, then Switch.
   Conditions are sampled the cycle they are added.
   AddStateCondition: must stay true in the state (else error -1).
   AddEntryCondition: checked only on the first cycle (bStateChanged).
   AddSwitchCondition: all must be true; Switch() is TRUE for one cycle.
   Timeout without switch -> error state -1.
   Typical: IF fbSM.Switch('Move', T#5S) THEN fbSM.SetNextState(nNext); *)
VAR_INPUT
	bTimeoutActive	: BOOL := TRUE;
	bStepMode		: BOOL := FALSE;
	bNextStep		: BOOL := FALSE;
	nStateForced	: INT := -1;
	hmiData			: REFERENCE TO ST_HMI_StateMachine;
	refLogger		: REFERENCE TO FB_Log;
END_VAR
VAR_OUTPUT
	bError			: BOOL;	// Error if state conditions are not TRUE or Timeout during to missing switch conditions.
	nErrorState		: INT := ERROR_STATE;	// the last state before error occured
	bSwitch			: BOOL;	// all switch conditions are TRUE
	bStateChanged	: BOOL;	// state has changed, TRUE for one cycle each state changing
	bStateValid		: BOOL;	// state conditions are true
	nState			: INT;	// current state, error = -1
	sState			: STRING;
	sTimeout		: STRING;
	tTimeInActState	: LTIME;	// Time in actual state
END_VAR
VAR

	//stStateHistory	: ARRAY[0..Settings.HISTORY_SIZE] OF ST_StateMachine_State;
	//better without struct, because of better debugging online view
	anStateHistory	: ARRAY[0..Parameter.HISTORY_SIZE] OF INT;
	asStateHistory	: ARRAY[0..Parameter.HISTORY_SIZE] OF STRING;
	
	tnTimeout		: TON;
	tnDelay			: TON;
	
	i					: INT;
	iState				: INT;
	iSwitch				: INT;
	iSwitchOrSection	: INT;
	
	nSwitchIndex		: INT;
	nStateIndex			: INT;
	
	abSwitchCondition	: ARRAY[0..Parameter.NUM_CON] OF BOOL;
	abStateCondition	: ARRAY[0..Parameter.NUM_CON] OF BOOL;
	asSwitchCondition	: ARRAY[0..Parameter.NUM_CON] OF T_MaxString;
	asStateCondition	: ARRAY[0..Parameter.NUM_CON] OF T_MaxString;
	
	nSwitchOrSection	: INT;	// 0 - global, 1..NUM_CON section
	anSwitchConSection	: ARRAY[0..Parameter.NUM_CON] OF INT;
	anOrSectionNextState	: ARRAY[0..Parameter.NUM_CON] OF INT;
	nOrSectionNextState	: INT;
	bOrSectionNextState	: BOOL;	// Oder-Sektion vorhanden
	bSwitchOr			: BOOL;
	
	bPreventErrorOverwrite	: BOOL;
	
	{attribute 'instance-path'}
	{attribute 'noinit'}
	instancePath: STRING;
	instanceName: STRING;	

	fbErrState		: FB_Alarm( TC_EVENTS.EventClassGeneral.E_StateCondition );
	fbErrSwitch		: FB_Alarm( TC_EVENTS.EventClassGeneral.E_SwitchCondition );
	
END_VAR
VAR CONSTANT
	ERROR_STATE	: INT := -1;	// ErrorState in Case of state conditions are not TRUE or switch timeout
END_VAR

METHOD PUBLIC AddEntryCondition : BOOL
VAR_INPUT
	bCondition:	BOOL;
	sName:		STRING;
END_VAR

// Must hold on the first cycle of a state (caller adds these before Switch).
// Later cycles: still record, but do not extra-fail.
IF bStateChanged THEN
	bStateValid R= NOT bCondition;
END_IF

IF iState <= Parameter.NUM_CON THEN
	abStateCondition[iState] := bCondition;
	asStateCondition[iState] := sName;
	iState := iState + 1;
END_IF
END_METHOD

METHOD PUBLIC AddStateCondition : BOOL
VAR_INPUT
	bCondition:	BOOL;
	sName:		STRING;
END_VAR

bStateValid R= NOT bCondition;

IF iState <= Parameter.NUM_CON THEN
	abStateCondition[iState] := bCondition;
	asStateCondition[iState] := sName;
	iState := iState + 1;
END_IF
END_METHOD

METHOD PUBLIC AddSwitchCondition : BOOL
VAR_INPUT
	bCondition:	BOOL;
	sName:		STRING;
END_VAR

bSwitch R= NOT bCondition OR NOT bStateValid;

IF iSwitch <= Parameter.NUM_CON THEN
	abSwitchCondition[iSwitch] := bCondition;
	asSwitchCondition[iSwitch] := sName;
	iSwitch := iSwitch + 1;
END_IF
END_METHOD

//FB_Init is always available implicitly and it is used primarily for initialization.
//The return value is not evaluated. For a specific influence, you can also declare the
//methods explicitly and provide additional code there with the standard initialization
//code. You can evaluate the return value.
METHOD FB_Init: BOOL
VAR_INPUT
    bInitRetains: BOOL; // TRUE: the retain variables are initialized (reset warm / reset cold)
    bInCopyCode: BOOL;  // TRUE: the instance will be copied to the copy code afterward (online change)   
END_VAR
VAR
	_i	: INT;
	_posDot	: INT;
	_instanceName: STRING;
END_VAR

_instanceName := instancePath;
FOR _i := 0 TO 9 DO
	_posDot := FIND( _instanceName, '.' );
	IF _posDot = 0 THEN
		EXIT;
	END_IF
	_instanceName := DELETE( _instanceName, _posDot, 1 );
END_FOR
SetInstanceName := _instanceName;
END_METHOD

METHOD PRIVATE FillRestOfConditions : BOOL
VAR_INPUT
END_VAR

// fill bits and empty strings in rest of state arrays
IF iState <= Parameter.NUM_CON THEN
	FOR i := iState TO Parameter.NUM_CON DO
		abStateCondition[i] := TRUE;
	END_FOR
	MemSet( ADR( asStateCondition[iState] ), 0, SIZEOF( asStateCondition[0] ) * TO_UINT( Parameter.NUM_CON - iState + 1 ) );
END_IF

// fill bits and empty strings in rest of switch arrays
IF iSwitch <= Parameter.NUM_CON THEN
	FOR i := iSwitch TO Parameter.NUM_CON DO
		abSwitchCondition[i] := TRUE;
		anSwitchConSection[i] := -1;
	END_FOR
	MemSet( ADR( asSwitchCondition[iSwitch] ), 0, SIZEOF( asSwitchCondition[0] ) * TO_UINT( Parameter.NUM_CON - iSwitch + 1 ) );
END_IF

// reset hmi data if available
IF __ISVALIDREF( hmiData ) THEN
	
	// fill bits and empty strings in rest of state arrays
	IF iState <= Parameter.NUM_CON THEN
		FOR i := iState TO Parameter.NUM_CON DO
			hmiData.stStateCondition[i].xState := TRUE;
			hmiData.stStateCondition[i].sName := '';
		END_FOR
	END_IF
	
	// fill bits and empty strings in rest of switch arrays
	IF iSwitch <= Parameter.NUM_CON THEN
		FOR i := iSwitch TO Parameter.NUM_CON DO
			hmiData.stSwitchCondition[i].xState := TRUE;
			hmiData.stSwitchCondition[i].sName := '';
		END_FOR
	END_IF
	
END_IF
END_METHOD

METHOD PUBLIC IncrementState : BOOL
VAR_INPUT
	nStateOffset:	INT;
END_VAR

SetNextState( nState + nStateOffset );
END_METHOD

METHOD PUBLIC Reset : BOOL
VAR_INPUT
END_VAR

bError := FALSE;
nErrorState := ERROR_STATE;
nState := 0;
sState := '';
sTimeout := '';
tTimeInActState := LTIME#0S;

// idle-ready: Switch() would trip error if bStateValid were FALSE
bSwitch := FALSE;
bStateValid := TRUE;
bStateChanged := FALSE;
bPreventErrorOverwrite := FALSE;

iState := 0;
iSwitch := 0;
iSwitchOrSection := 0;

tnTimeout( IN := FALSE );
tnDelay( IN := FALSE );

FOR i := 0 TO Parameter.HISTORY_SIZE DO
	anStateHistory[i] := 0;
	asStateHistory[i] := '';
	IF __ISVALIDREF( hmiData ) THEN
		hmiData.stStateHistory[i].nState := 0;
		hmiData.stStateHistory[i].sState := '';
	END_IF
END_FOR

MEMSET( ADR( abSwitchCondition ), 0, SIZEOF( abSwitchCondition ) );
MEMSET( ADR( abStateCondition ), 0, SIZEOF( abStateCondition ) );
MEMSET( ADR( asSwitchCondition ), 0, SIZEOF( asSwitchCondition ) );
MEMSET( ADR( asStateCondition ), 0, SIZEOF( asStateCondition ) );

IF __ISVALIDREF( hmiData ) THEN
	hmiData.nState := 0;
	hmiData.sState := '';
END_IF
END_METHOD

METHOD PRIVATE SaveStateHistory : BOOL
VAR_INPUT
	nState:	INT;
END_VAR

IF __ISVALIDREF(refLogger) THEN
	refLogger.AppendStringToLine( instanceName );
	refLogger.AppendStringToLine( ' - [' );
	refLogger.AppendStringToLine( INT_TO_STRING( nState ) );
	refLogger.AppendStringToLine( '] - ' );
	refLogger.AppendStringToLine( sState );
	refLogger.LogLine();
END_IF

FOR i := Parameter.HISTORY_SIZE-1 TO 0 BY -1 DO
	anStateHistory[i+1] := anStateHistory[i];
	asStateHistory[i+1] := asStateHistory[i];
	IF __ISVALIDREF( hmiData ) THEN
		hmiData.stStateHistory[i+1].nState := anStateHistory[i];
		hmiData.stStateHistory[i+1].sState := asStateHistory[i];
	END_IF
END_FOR

anStateHistory[0] := nState;
asStateHistory[0] := '';
IF __ISVALIDREF( hmiData ) THEN
	hmiData.stStateHistory[0].nState := nState;
	hmiData.stStateHistory[0].sState := '';
END_IF
END_METHOD

METHOD PUBLIC SetError : BOOL
VAR_INPUT
END_VAR

bError := TRUE;
IF nState <> ERROR_STATE THEN
	bPreventErrorOverwrite := TRUE;
	nErrorState := nState;
	SetNextState( ERROR_STATE );
	sState := 'Error';
END_IF
END_METHOD

PROPERTY PUBLIC SetInstanceName : STRING
SET
instanceName := SetInstanceName;
END_SET
END_PROPERTY

METHOD PUBLIC SetNextState : BOOL
VAR_INPUT
	nNextState:	INT;
END_VAR

nState := nNextState;
bStateChanged := TRUE;

// Reset validation data
bStateValid := TRUE;

saveStateHistory( nNextState );
END_METHOD

METHOD PUBLIC Switch : BOOL
VAR_INPUT
	sName		: STRING;
	tTimeout	: TIME;
END_VAR

// timeout monitoring
IF tTimeout <> T#0S THEN
	tnTimeout(
		IN := NOT bSwitch,
		PT := tTimeout
	);
	sTimeout := TIME_TO_STRING( tnTimeout.ET );
	IF tnTimeout.Q THEN
		fbErrSwitch.setEventWithOneArgument( TRUE, sName );
		setNextState( -1 );	// error
		bError := TRUE;
	END_IF
ELSE
	tnTimeout( IN := FALSE );
	sTimeout := TIME_TO_STRING( tTimeout );
END_IF

// state monitoring
IF NOT bStateValid THEN
	fbErrState.setEventWithOneArgument( TRUE, sName );
	setNextState( -1 );	// error
	bError := TRUE;
END_IF

switch := bSwitch;

sState := sName;

IF bStateChanged THEN
	FillRestOfConditions();
END_IF

// reset i's
iState := 0;
iSwitch := 0;

// reset switch info for next cycle
bSwitch := TRUE;
bStateValid := TRUE;

// switch is only one cycle active, reset switch info
bStateChanged := FALSE;
END_METHOD

METHOD PUBLIC SwitchWithDelay : BOOL
VAR_INPUT
	sName:	STRING;
	tTimeout:	TIME;
	tDelayTime:	TIME;	// state is active at least this time, after all switch conditions are TRUE
END_VAR
// timeout monitoring
IF tDelayTime <> T#0S THEN
	tnDelay(
		IN := bSwitch,
		PT := tDelayTime
	);
	IF NOT tnDelay.Q THEN
		bSwitch := FALSE;
	END_IF
ELSE
	tnDelay( IN := FALSE );
END_IF

IF tTimeout <> T#0S THEN
	tTimeout := tTimeout + tDelayTime;
END_IF

switchWithDelay := switch( sName := sName, tTimeout := tTimeout ) ;

IF switchWithDelay THEN
	tnDelay( IN := FALSE );
END_IF
END_METHOD

END_FUNCTION_BLOCK

// ---- EventLogger/Logger/FB_Log.TcPOU
FUNCTION_BLOCK FB_Log
VAR_INPUT
	refTimeStamp	: REFERENCE TO ST_SysTime;
END_VAR
VAR_OUTPUT
	xBusy		: BOOL;
	xBufferFull	: BOOL;
END_VAR
VAR
	fbFileOpen		: FB_FileOpen;
	fbFileRead		: FB_FileRead;
	fbFileWrite		: FB_FileWrite;
	fbFileClose		: FB_FileClose;
	fileHandle		: UINT;

	// file variables
	filePath		: STRING := 'debug.log';
	nStringIndexTemp: INT;
	nStringIndex	: INT;
	nStringPointer	: INT;
	sLineToWrite	: ARRAY[0..MAX_STRINGS] OF STRING( Parameter.MAX_STRING_LENGTH );
	
	xNewLine		: BOOL;
	
    stateFile	: FB_StateMachine;

END_VAR
VAR CONSTANT
	MAX_STRINGS		: INT := 99;
END_VAR


CASE stateFile.nState OF
	
	-1:	// Error
		IF stateFile.bStateChanged THEN
			xBusy := FALSE;
			fbFileOpen( bExecute := FALSE );
			fbFileRead( bExecute := FALSE );
			fbFileWrite( bExecute := FALSE );
			fbFileClose( bExecute := FALSE );
			nStringIndex := 0;
			nStringPointer := 0;
		END_IF
		
		xNewLine := nStringIndex <> nStringPointer;
		
		stateFile.AddSwitchCondition( NOT xNewLine, '' );
		IF stateFile.Switch( 'Error', T#0S ) THEN
			stateFile.Reset();
		END_IF
	
	0: // Initialisierung
		stateFile.AddSwitchCondition( xNewLine, '' );
		
		IF stateFile.Switch( 'Init', T#0S ) THEN
			xBusy := TRUE;
			fbFileOpen( bExecute := FALSE );
			fbFileRead( bExecute := FALSE );
			fbFileWrite( bExecute := FALSE );
			fbFileClose( bExecute := FALSE );
			stateFile.IncrementState( 1 );
		END_IF;
	
	1: // open file
		fbFileOpen(
			bExecute := TRUE,
			nMode := FOPEN_MODEAPPEND,
			sPathName := filePath,
			hFile => fileHandle
		);
		
		stateFile.AddSwitchCondition( fileHandle <> 0 OR fbFileOpen.bError, '' );
		
		IF stateFile.Switch( 'Open File', T#0S ) THEN
			IF fileHandle <> 0 THEN
				stateFile.IncrementState( 1 );
			END_IF
			IF fbFileOpen.bError THEN
				stateFile.SetError();
			END_IF
		END_IF
	
	2: // Zeile an Datei anfügen
		fbFileWrite(
			bExecute := TRUE,
			hFile := fileHandle,
			pWriteBuff := ADR( sLineToWrite[nStringPointer] ),
			cbWriteLen := INT_TO_UINT( LEN( sLineToWrite[nStringPointer] ) )
		);
		
		stateFile.AddSwitchCondition( NOT fbFileWrite.bBusy OR fbFileWrite.bError, '' );
		
		IF stateFile.Switch( 'Write File', T#0S ) THEN
			IF NOT fbFileWrite.bError THEN
				sLineToWrite[nStringPointer] := '';
				Increment( nStringPointer );
				IF xNewLine THEN
					stateFile.SetNextState( 2 );
				ELSE
					stateFile.IncrementState( 1 );
				END_IF
			ELSE
				stateFile.SetError();
			END_IF
			fbFileWrite( bExecute := FALSE );
		END_IF

	3: // Datei schließen
		fbFileClose(
			bExecute := TRUE,
			hFile := fileHandle
		);
		stateFile.AddSwitchCondition( NOT fbFileClose.bBusy OR fbFileClose.bError, '' );
		IF stateFile.Switch( 'Close File', T#0S ) THEN
			
			fbFileOpen( bExecute := FALSE );
			fbFileRead( bExecute := FALSE );
			fbFileWrite( bExecute := FALSE );
			fbFileClose( bExecute := FALSE );
			
			xBusy := FALSE;
			fileHandle := 0;
			fbFileClose.bExecute := FALSE;
			stateFile.SetNextState( 0 );
		END_IF
		
END_CASE

METHOD PUBLIC AppendStringToLine : BOOL	// REFRENCE TO FB_Log
VAR_INPUT
	sNewString	: STRING( Parameter.MAX_STRING_LENGTH );
END_VAR

sLineToWrite[nStringIndex] := CONCAT( sLineToWrite[nStringIndex], sNewString );
//AppendStringToLine := THIS^;
END_METHOD

METHOD PRIVATE Increment : INT
VAR_IN_OUT
	nValue	: INT;
END_VAR

IF nValue >= MAX_STRINGS THEN
	nValue := 0;
ELSE
	nValue := nValue + 1;
END_IF

xNewLine := nStringIndex <> nStringPointer;
END_METHOD

METHOD PUBLIC LogDate : BOOL
VAR_INPUT
END_VAR
VAR
	nLen	: INT := 0;
END_VAR

AppendStringToLine( refTimeStamp.sDate );
LogLineNoTime();
END_METHOD

METHOD PUBLIC LogLine : BOOL
VAR_INPUT
END_VAR
VAR
	nLen	: INT := 0;
END_VAR

IF __ISVALIDREF( refTimeStamp ) THEN
	nLen := LEN( refTimeStamp.sTimestamp );
END_IF

IF LEN( sLineToWrite[nStringIndex] ) > ( UDINT_TO_DINT( Parameter.MAX_STRING_LENGTH ) - ( nLen + 4 ) ) THEN
	DELETE( sLineToWrite[nStringIndex], ( nLen + 4 ), LEN( sLineToWrite[nStringIndex] ) - ( nLen + 4 - 1 ) );
	AppendStringToLine( '>>' );
END_IF

AppendStringToLine( '$R$N' );

IF __ISVALIDREF( refTimeStamp ) THEN
	sLineToWrite[nStringIndex] := CONCAT( ' ', sLineToWrite[nStringIndex] );
	sLineToWrite[nStringIndex] := CONCAT( refTimeStamp.sTimestamp, sLineToWrite[nStringIndex] );
END_IF

Increment( nStringIndex );
IF sLineToWrite[nStringIndex] <> '' THEN
	sLineToWrite[nStringIndex] := '!!! Buffer Overload !!!';
	AppendStringToLine( '$R$N' );
END_IF
END_METHOD

METHOD PUBLIC LogLineNoTime : BOOL
VAR_INPUT
END_VAR
VAR
	nLen	: INT := 0;
END_VAR

IF LEN( sLineToWrite[nStringIndex] ) > ( UDINT_TO_DINT( Parameter.MAX_STRING_LENGTH ) - ( nLen + 4 ) ) THEN
	DELETE( sLineToWrite[nStringIndex], ( nLen + 4 ), LEN( sLineToWrite[nStringIndex] ) - ( nLen + 4 - 1 ) );
	AppendStringToLine( '>>' );
END_IF

AppendStringToLine( '$R$N' );

Increment( nStringIndex );
IF sLineToWrite[nStringIndex] <> '' THEN
	sLineToWrite[nStringIndex] := '!!! Buffer Overload !!!';
END_IF
END_METHOD

METHOD PUBLIC SetFilePath : BOOL
VAR_INPUT
	sFilePath	: STRING;
END_VAR

filePath := sFilePath;
END_METHOD

ACTION TODO:
(*

- file size überwachen und zu große Dateien verhindern
- Option zu neuer Datei mit Zeitstempel

*)
END_ACTION

END_FUNCTION_BLOCK

// ---- EventLogger/EventListenerExtV2/FB_EventListenerExtV2.TcPOU
FUNCTION_BLOCK FB_EventListenerExtV2 EXTENDS FB_ListenerBase2 IMPLEMENTS I_EventListener
VAR_INPUT
    bInsertFirst : BOOL := TRUE;
    aEventClasses: ARRAY[1..Parameter.nMaxEventClasses] OF GUID;
END_VAR
VAR
	ipMessageFilterConfig : ITcEventFilterConfig;
	ipAlarmFilterConfig : ITcEventFilterConfig;
	hrFilterConfig : HRESULT;
END_VAR
VAR_OUTPUT
    aEventEntryTable: ARRAY[0..Parameter.nMaxEventEntries] OF ST_EventEntryTableListener;
    aEvents : ARRAY[1..80] OF ST_ReadEvent; // Legacy Event Table 
END_VAR
VAR
	bEventEntryTableTestandSet : BOOL;
    fbGetTimeZoneInformation: FB_GetTimeZoneInformation;
END_VAR
VAR
    nCounter : DINT;
    stSeverestAlarmEntryTable:  ST_EventEntryTableListener;
    stLastEventEntryTable:  ST_EventEntryTableListener; 
END_VAR
VAR
    nLanguage: INT := 1033;
    sLanguage: STRING := 'en';
    bChangeLanguageInterlock : BOOL;
END_VAR
VAR	 // Visu variables --- Legacy...
	nVisuTableIndex : INT := 0;
	bVisuIndexingPlus: BOOL;
	bVisuIndexingMinus: BOOL;

	bVisuDisableIndexingPlus: BOOL;
	bVisuDisableIndexingMinus: BOOL;
    bCmdDeleteEventsFromTableHmi: BOOL; // HMI
END_VAR

METHOD PRIVATE ChangeLanguage : HRESULT
VAR
    hr : HRESULT;
    UTF8 : STRING(255);
END_VAR
VAR_INST
    {attribute 'no_copy'}
    fbRequestText : FB_RequestEventText;
    {attribute 'no_copy'}
    fbRequestClassName : FB_RequestEventClassName;
END_VAR
VAR_INST
    stEventEntryTemp: ST_EventEntryTableListener;
END_VAR
VAR_INST
    nStep : E_AlarmMessage;
    nStepRequestText : E_AlarmMessage := E_AlarmMessage.Done;
    nStepRequestClass : E_AlarmMessage := E_AlarmMessage.Done;
END_VAR
VAR_INST
    nTranslated : DINT;
END_VAR
VAR
    nEntryIndex : DINT;
END_VAR
    ChangeLanguage := E_FAIL;
    
    bChangeLanguageInterlock := TRUE;
	
// Fast Case of nStep
    // CASE: E_AlarmMessage.RequestText
    IF nStep = E_AlarmMessage.RequestText THEN
        
        stEventEntryTemp := aEventEntryTable[nTranslated];
        nStepRequestText := E_AlarmMessage.RequestText;
        nStepRequestClass := E_AlarmMessage.RequestText;
        nStep := E_AlarmMessage.ReceiveText;
	END_IF
    // CASE: E_AlarmMessage.ReceiveText
    IF nStep = E_AlarmMessage.ReceiveText THEN
        IF nStepRequestText = E_AlarmMessage.Done AND
           nStepRequestClass = E_AlarmMessage.Done THEN
           nStep := E_AlarmMessage.Insert;
		END_IF
	END_IF
    // CASE: E_AlarmMessage.Insert
    IF nStep = E_AlarmMessage.Insert THEN
        
            nEntryIndex := GetIndex(stEventEntryTemp, FALSE);
            IF nEntryIndex >= 0 THEN
                IF stEventEntryTemp.sText <> '{0}' AND stEventEntryTemp.sText <> '' THEN
                    aEventEntryTable[nEntryIndex].sText := stEventEntryTemp.sText;
				END_IF
                IF stEventEntryTemp.EventClassName <> '{0}' AND stEventEntryTemp.EventClassName <> '' THEN
                    aEventEntryTable[nEntryIndex].EventClassName := stEventEntryTemp.EventClassName;
				END_IF
            END_IF
            stSeverestAlarmEntryTable:=  GetSeverestAlarmEntryTable();
            stLastEventEntryTable:=  GetLastEventEntryTable(); 
            UpdateLegacyTable();
            
            nStep := E_AlarmMessage.Done;
	END_IF
    // CASE: Done   
    IF nStep = E_AlarmMessage.Done THEN
        nTranslated := nTranslated + 1;
            IF nTranslated > nCounter THEN
                  nTranslated := 0;
                  ChangeLanguage := S_OK;
                  bChangeLanguageInterlock := FALSE;
            END_IF
            nStep := E_AlarmMessage.RequestText;
            MEMSET(destAddr:= ADR(stEventEntryTemp), fillByte := 16#00 , n:= SIZEOF(stEventEntryTemp));
	END_IF     


// Fast Case of nStepRequestText
    // CASE: RequestText   
    IF nStepRequestText = E_AlarmMessage.RequestText THEN
        fbRequestText.Request( eventClass:=stEventEntryTemp.EventClass, nEventId:=stEventEntryTemp.nEventId, nLangId:=LangId, ipArgs:=stEventEntryTemp.ipArguments );
        nStepRequestText := E_AlarmMessage.ReceiveText; 
	END_IF
    // CASE: ReceiveText   
    IF nStepRequestText = E_AlarmMessage.ReceiveText THEN
        IF NOT fbRequestText.bBusy AND NOT fbRequestText.bError THEN
            fbRequestText.GetString(UTF8, SIZEOF(UTF8));
            UTF8_TO_STRING(pDstSTRING:=ADR(stEventEntryTemp.sText) , pSrcUTF8:=ADR(UTF8) , nDstSize:=SIZEOF(stEventEntryTemp.sText) , nDstLen=> );
            nStepRequestText := E_AlarmMessage.Done;
        ELSIF fbRequestText.bError THEN 
            nStepRequestText := E_AlarmMessage.RequestText;
        END_IF 
	END_IF
 
// Fast Case of nStepRequestClass
    // CASE: RequestText   
    IF nStepRequestClass = E_AlarmMessage.RequestText THEN
        fbRequestClassName.Request(eventClass:=stEventEntryTemp.EventClass, nLangId:=LangId,);
        nStepRequestClass := E_AlarmMessage.ReceiveText;
	END_IF
    // CASE: ReceiveText   
    IF nStepRequestClass = E_AlarmMessage.ReceiveText THEN
        IF NOT fbRequestClassName.bBusy AND NOT fbRequestClassName.bError THEN
            fbRequestClassName.GetString(UTF8, SIZEOF(UTF8));
            UTF8_TO_STRING(pDstSTRING:=ADR(stEventEntryTemp.EventClassName) , pSrcUTF8:=ADR(UTF8) , nDstSize:=SIZEOF(stEventEntryTemp.EventClassName) , nDstLen=> );
            nStepRequestClass := E_AlarmMessage.Done;
        ELSIF fbRequestClassName.bError THEN 
            nStepRequestClass := E_AlarmMessage.RequestText;
        END_IF
	END_IF
END_METHOD

METHOD PRIVATE DeleteEntryFromEventTable : HRESULT
VAR_INPUT
	index: UDINT;
END_VAR

IF NOT ( index >= 0 AND TO_DINT(index) <= Parameter.nMaxEventEntries ) THEN
	DeleteEntryFromEventTable := E_FAIL;
	RETURN;
END_IF

MEMSET( destAddr := ADR(aEventEntryTable[index]), fillByte := 16#00, n := SIZEOF(aEventEntryTable[index]) );
IF MEMMOVE( srcAddr := ADR(aEventEntryTable[index + 1]), destAddr := ADR(aEventEntryTable[index]), n := ( SIZEOF(aEventEntryTable) - SIZEOF(aEventEntryTable[0]) * ( index + 1 ) ) ) <= 0 THEN
	DeleteEntryFromEventTable := E_FAIL;
	RETURN;
ELSE
	MEMSET( destAddr := ADR(aEventEntryTable[Parameter.nMaxEventEntries]), fillByte := 16#00, n := SIZEOF(aEventEntryTable[Parameter.nMaxEventEntries]) );
	nCounter := LIMIT( 0, nCounter - 1, TO_DINT(Parameter.nMaxEventEntries) );
END_IF

stSeverestAlarmEntryTable := GetSeverestAlarmEntryTable();
stLastEventEntryTable := GetLastEventEntryTable();
UpdateLegacyTable();
END_METHOD

METHOD PUBLIC DeleteEventsFromTable : BOOL
VAR_INPUT
END_VAR
VAR_INST
	i: DINT;
END_VAR

IF TestandSet(bEventEntryTableTestandSet) THEN
	IF NOT bChangeLanguageInterlock THEN
		FOR i := 0 TO Parameter.nMaxEventEntries BY 1 DO
			IF aEventEntryTable[i].nEventId <> 0
			AND aEventEntryTable[i].bIsEvent THEN
				DeleteEntryFromEventTable(DINT_TO_UDINT(i));
				i := i-1;
			ELSIF aEventEntryTable[i].nEventId = 0 THEN
				EXIT;
			END_IF
		END_FOR
	END_IF
bEventEntryTableTestandSet := FALSE;
END_IF
END_METHOD

METHOD Execute : HRESULT
VAR_INST
    nLanguangeTemp : INT := nLanguage;
    hrs : HRESULT := S_OK;
END_VAR
VAR_INST
    bGetTimeZone : BOOL := TRUE;
END_VAR

Execute := SUPER^.Execute(); //retrieve events

HMI();

IF bGetTimeZone THEN
   bGetTimeZone := FALSE;
   fbGetTimeZoneInformation( bExecute := TRUE );
ELSE
   fbGetTimeZoneInformation( bExecute := FALSE );        
END_IF

IF nLanguangeTemp <> nLanguage OR hrs <> S_OK THEN
	IF TestandSet(bEventEntryTableTestandSet) THEN
		nLanguangeTemp := nLanguage;
		hrs := ChangeLanguage();
		bEventEntryTableTestandSet := FALSE;
	END_IF
END_IF
END_METHOD

PROPERTY PUBLIC FlagInsertFirst : BOOL
GET
FlagInsertFirst := bInsertFirst;
END_GET
SET
bInsertFirst := FlagInsertFirst;
END_SET
END_PROPERTY

METHOD PUBLIC GetEventByIndex : HRESULT
    VAR_OUTPUT
        sTimestamp: STRING(80); // 
        sTimestampConfirmed: STRING(80);
        sTimestampCleared: STRING(80);
        sText: STRING(255); //
        sSourceName: STRING(255); //
        EventClassName: STRING(255); //
        eConfirmationState : BYTE;
        eSeverity :  BYTE; // INT
    END_VAR
VAR_INPUT
    nIndex : UDINT;
END_VAR
IF nIndex >= 1 AND nIndex <= TO_UDINT(Parameter.nMaxEventEntries) THEN
        sTimestamp := aEventEntryTable[nIndex].sTimestamp;
        sTimestampConfirmed := aEventEntryTable[nIndex].sTimestampConfirmed;
        sTimestampCleared := aEventEntryTable[nIndex].sTimestampCleared;
        sText := aEventEntryTable[nIndex].sText; //
        sSourceName:= aEventEntryTable[nIndex].sSourceName;
        EventClassName := aEventEntryTable[nIndex].EventClassName;
        eConfirmationState := TO_BYTE(aEventEntryTable[nIndex].eConfirmationState);
        eSeverity := TO_BYTE(aEventEntryTable[nIndex].eSeverity);
        
        GetEventByIndex := S_OK;
ELSE
        GetEventByIndex := E_FAIL;
END_IF
END_METHOD

METHOD PRIVATE GetIndex : DINT
VAR_INPUT
	stEventEntryTableTemp: ST_EventEntryTableListener;
	bWithTimeStamp: BOOL;
END_VAR
VAR
	i: DINT;
END_VAR

GetIndex := -1;
FOR i := 0 TO TO_DINT(Parameter.nMaxEventEntries) BY 1 DO
	IF aEventEntryTable[i].nEventId = stEventEntryTableTemp.nEventId
	AND_THEN aEventEntryTable[i].eSeverity = stEventEntryTableTemp.eSeverity
	AND_THEN MEMCMP( ADR( aEventEntryTable[i].EventClass ), ADR( stEventEntryTableTemp.EventClass ), SIZEOF( stEventEntryTableTemp.EventClass ) ) = 0
	AND_THEN aEventEntryTable[i].sSourceName = stEventEntryTableTemp.sSourceName THEN
		IF bWithTimeStamp THEN 
			IF aEventEntryTable[i].sTimestamp = stEventEntryTableTemp.sTimestamp THEN
				GetIndex := i;
			END_IF
		END_IF
			GetIndex := i;
		EXIT;
	END_IF
END_FOR
END_METHOD

METHOD PRIVATE GetLastEventEntryTable : ST_EventEntryTableListener
VAR_INPUT
END_VAR

IF bInsertFirst THEN
    GetLastEventEntryTable := aEventEntryTable[0];
ELSE
    GetLastEventEntryTable := aEventEntryTable[LIMIT( 0, nCounter - 1, Parameter.nMaxEventEntries)];
END_IF
END_METHOD

METHOD PRIVATE GetSeverestAlarmEntryTable : ST_EventEntryTableListener
VAR_INPUT
END_VAR
VAR
    i : DINT;
END_VAR
IF bInsertFirst THEN
    FOR i := TO_DINT(LIMIT( 0, (nCounter - 1), TO_DINT(Parameter.nMaxEventEntries))) TO 0 BY (- 1) DO
        IF aEventEntryTable[i].bIsAlarm AND NOT GetSeverestAlarmEntryTable.bIsAlarm THEN
            GetSeverestAlarmEntryTable := aEventEntryTable[i];
        ELSIF aEventEntryTable[i].eSeverity >= GetSeverestAlarmEntryTable.eSeverity THEN
            GetSeverestAlarmEntryTable := aEventEntryTable[i];
        END_IF
    END_FOR  
ELSE
    FOR i := 0 TO TO_DINT(LIMIT( 0, (nCounter - 1), TO_DINT(Parameter.nMaxEventEntries))) DO
        IF aEventEntryTable[i].bIsAlarm AND NOT GetSeverestAlarmEntryTable.bIsAlarm THEN
            GetSeverestAlarmEntryTable := aEventEntryTable[i];
        ELSIF aEventEntryTable[i].eSeverity >= GetSeverestAlarmEntryTable.eSeverity THEN
            GetSeverestAlarmEntryTable := aEventEntryTable[i];
        END_IF
    END_FOR 
END_IF
END_METHOD

METHOD PRIVATE HMI : BOOL
VAR_INST
    nCounterTemp : DINT;
    trigVisuIndexingPlus: R_TRIG;
	trigVisuIndexingMinus: R_TRIG;
    trigDeleteEventsFromTabl: R_TRIG;
END_VAR
IF nCounterTemp <> nCounter THEN
    nCounterTemp := nCounter;
    nVisuTableIndex := 0;
END_IF

IF nVisuTableIndex <= nCounter - Parameter.nNUM_OF_MESSAGES_VISU
AND nCounter > Parameter.nNUM_OF_MESSAGES_VISU
AND nVisuTableIndex < UINT_TO_INT( Parameter.nMaxEventEntries ) THEN
	bVisuDisableIndexingPlus := FALSE;
ELSE
	bVisuDisableIndexingPlus := TRUE;
END_IF

IF nVisuTableIndex > 0 THEN
	bVisuDisableIndexingMinus := FALSE;
ELSE
	bVisuDisableIndexingMinus := TRUE;
END_IF

trigVisuIndexingPlus( clk := bVisuIndexingPlus );
IF trigVisuIndexingPlus.Q THEN
	nVisuTableIndex := nVisuTableIndex + 1;
END_IF

trigVisuIndexingMinus( clk := bVisuIndexingMinus );
IF trigVisuIndexingMinus.Q THEN
	nVisuTableIndex := nVisuTableIndex - 1;
END_IF

trigDeleteEventsFromTabl( CLK := bCmdDeleteEventsFromTableHmi );
IF trigDeleteEventsFromTabl.Q THEN
	DeleteEventsFromTable();
END_IF
END_METHOD

METHOD Initialize : HRESULT
VAR_INPUT
END_VAR
VAR
    i : UINT;
END_VAR

hrFilterConfig := THIS^.Unsubscribe();
hrFilterConfig := THIS^.Subscribe( ADR(ipMessageFilterConfig), ADR(ipAlarmFilterConfig) );

IF ( ipMessageFilterConfig <> 0 ) AND hrFilterConfig = S_OK THEN
	FOR i := 1 TO Parameter.nMaxEventClasses DO 
        IF MEMCMP( ADR(aEventClasses[i]), ADR(EMPTY_GUID_STRUCT), SIZEOF(EMPTY_GUID_STRUCT) ) > 0 THEN
            ipMessageFilterConfig.AddEventClass( aEventClasses[i], TcEventSeverity.Verbose );
        END_IF
    END_FOR
END_IF

IF ( ipAlarmFilterConfig <> 0 ) AND hrFilterConfig = S_OK THEN
	FOR i := 1 TO Parameter.nMaxEventClasses DO 
        IF MEMCMP( ADR(aEventClasses[i]), ADR(EMPTY_GUID_STRUCT), SIZEOF(EMPTY_GUID_STRUCT) ) > 0 THEN
            ipAlarmFilterConfig.AddEventClass( aEventClasses[i], TcEventSeverity.Verbose );
        END_IF
    END_FOR
END_IF
END_METHOD

METHOD PRIVATE Insert : HRESULT
VAR_INPUT
    stEventEntryTable: ST_EventEntryTableListener;
END_VAR
IF bInsertFirst THEN
    Insert := InsertFirst(stEventEntryTable := stEventEntryTable);
ELSE
    Insert := InsertLast(stEventEntryTable := stEventEntryTable);
END_IF
    stSeverestAlarmEntryTable:=  GetSeverestAlarmEntryTable();
    stLastEventEntryTable:=  GetLastEventEntryTable();
    UpdateLegacyTable();
END_METHOD

METHOD PRIVATE InsertFirst : HRESULT
VAR_INPUT
    stEventEntryTable: ST_EventEntryTableListener;
END_VAR
IF Parameter.nMaxEventEntries <= 0 THEN
	InsertFirst := E_FAIL;
	RETURN;
END_IF

InsertFirst := E_FAIL;

nCounter := nCounter + 1;
IF nCounter > TO_DINT(Parameter.nMaxEventEntries) THEN
	nCounter := TO_DINT(Parameter.nMaxEventEntries);
END_IF

IF MEMMOVE(srcAddr := ADR(aEventEntryTable[0]), destAddr := ADR(aEventEntryTable[1]), n := (SIZEOF(aEventEntryTable)- SIZEOF(aEventEntryTable[0]))) <= 0 THEN
	InsertFirst := E_FAIL;
	RETURN;
END_IF
aEventEntryTable[0] := stEventEntryTable;

InsertFirst := S_OK;
END_METHOD

METHOD PRIVATE InsertLast : HRESULT
VAR_INPUT
    stEventEntryTable: ST_EventEntryTableListener;
END_VAR
IF Parameter.nMaxEventEntries <= 0 THEN
	InsertLast := E_FAIL;
	RETURN;
END_IF

InsertLast := E_FAIL;

nCounter := nCounter + 1;
IF (nCounter - 1) <= TO_DINT(Parameter.nMaxEventEntries) THEN
	aEventEntryTable[nCounter-1] := stEventEntryTable;   
ELSE
	IF MEMMOVE(srcAddr := ADR(aEventEntryTable[1]), destAddr := ADR(aEventEntryTable[0]), n := (SIZEOF(aEventEntryTable)-SIZEOF(aEventEntryTable[0]))) <= 0 THEN
		InsertLast := E_FAIL;
		RETURN;
	END_IF
	aEventEntryTable[Parameter.nMaxEventEntries] := stEventEntryTable;
    nCounter := TO_DINT(Parameter.nMaxEventEntries);
END_IF

InsertLast := S_OK;
END_METHOD

METHOD PUBLIC isErrorRaised : BOOL
VAR_INPUT
	nZoneIdToCheck	: UDINT;
END_VAR
VAR
	i	: UINT;
END_VAR

isErrorRaised := FALSE;
FOR i := 0 TO Parameter.nMaxEventEntries BY 1 DO
	IF aEventEntryTable[i].nSourceId = nZoneIdToCheck
	AND aEventEntryTable[i].bIsAlarm THEN
		isErrorRaised := TRUE;
		EXIT;
	END_IF
END_FOR
END_METHOD

PROPERTY PUBLIC LangId : INT
GET
LangId := nLanguage;
END_GET
SET
nLanguage := LangId;
END_SET
END_PROPERTY

METHOD PUBLIC LanguageId : HRESULT
VAR_INPUT
	sCurrentLanguage	: STRING;
END_VAR

// Set language
IF sLanguage <> sCurrentLanguage THEN
	IF sCurrentLanguage = 'de' OR sCurrentLanguage = 'DE' THEN
		LangId := 1031;
	ELSIF sCurrentLanguage = 'en' OR sCurrentLanguage = 'EN' OR sCurrentLanguage = 'gb' OR sCurrentLanguage = 'GB' THEN
		LangId := 1033;
	ELSIF sCurrentLanguage = 'cz' OR sCurrentLanguage = 'CZ' THEN
		LangId := 1029;
	END_IF
	sLanguage := sCurrentLanguage;
END_IF
END_METHOD

PROPERTY PUBLIC LastEventEntryTable : ST_EventEntryTableListener
GET
LastEventEntryTable := stLastEventEntryTable;
END_GET
END_PROPERTY

PROPERTY PUBLIC NumberActiveEvents : UDINT;
GET
NumberActiveEvents := TO_UDINT(nCounter);
END_GET
END_PROPERTY

METHOD OnAlarmCleared : HRESULT
VAR_INPUT
	fbEvent : REFERENCE TO FB_TcEvent;
END_VAR
VAR
    hr : HRESULT;
    UTF8 : STRING(255);
END_VAR
VAR_INST
    {attribute 'no_copy'}
    fbRequestText : FB_RequestEventText;
    {attribute 'no_copy'}
    fbRequestClassName : FB_RequestEventClassName;
END_VAR
VAR_INST
    stEventEntryTemp: ST_EventEntryTableListener;
END_VAR
VAR_INST
    nStep : E_AlarmMessage;
    nStepRequestText : E_AlarmMessage := E_AlarmMessage.Done;
    nStepRequestClass : E_AlarmMessage := E_AlarmMessage.Done;
	
	nCounterNothingFound : DINT;
END_VAR
VAR
    nEntryIndex : DINT;
END_VAR

IF NOT __ISVALIDREF(fbEvent) THEN
	RETURN;
ELSE
	OnAlarmCleared := E_FAIL; // in order to receive more callbacks (Set <> S_OK in order to cancel the callbacks for this program cycle.)
	IF bChangeLanguageInterlock THEN
		RETURN;
	END_IF    
END_IF

// Fast Case of nStep
    // CASE: E_AlarmMessage.RequestText
    
    IF nStep = E_AlarmMessage.RequestText THEN
        nStepRequestText := E_AlarmMessage.RequestText;
        nStepRequestClass := E_AlarmMessage.RequestText;
        nStep := E_AlarmMessage.ReceiveText;
	END_IF
    // CASE: E_AlarmMessage.ReceiveText
    IF nStep = E_AlarmMessage.ReceiveText THEN
        IF nStepRequestText = E_AlarmMessage.Done AND
           nStepRequestClass = E_AlarmMessage.Done THEN
           nStep := E_AlarmMessage.Insert;
		END_IF
	END_IF
    // CASE: E_AlarmMessage.Insert
    IF nStep = E_AlarmMessage.Insert THEN
        
            stEventEntryTemp.sSourceName := fbEvent.ipSourceInfo.sName;
			stEventEntryTemp.nSourceId := fbEvent.ipSourceInfo.nId;
            stEventEntryTemp.eSeverity := fbEvent.eSeverity;
            IF stEventEntryTemp.eSeverity = 0 THEN stEventEntryTemp.sSeverity := 'Verbose';
            ELSIF stEventEntryTemp.eSeverity = 1 THEN stEventEntryTemp.sSeverity := 'Info';
            ELSIF stEventEntryTemp.eSeverity = 2 THEN stEventEntryTemp.sSeverity := 'Warning';
            ELSIF stEventEntryTemp.eSeverity = 3 THEN stEventEntryTemp.sSeverity := 'Error';
            ELSIF stEventEntryTemp.eSeverity = 4 THEN stEventEntryTemp.sSeverity := 'Critical'; END_IF
            stEventEntryTemp.EventClass := fbEvent.EventClass;
            stEventEntryTemp.nEventId := fbEvent.nEventId;
            stEventEntryTemp.ipArguments := fbEvent.ipArguments;
            
			IF TestandSet(bEventEntryTableTestandSet) THEN	
            nEntryIndex := GetIndex(stEventEntryTemp, FALSE);
            IF nEntryIndex >= 0 THEN

                aEventEntryTable[nEntryIndex].bLogged := FALSE;
                aEventEntryTable[nEntryIndex].eConfirmationState := TcEventConfirmationState.Reset;
                aEventEntryTable[nEntryIndex].sTimestampLog := SYSTEMTIME_TO_STRING(UlintToSystemTime(fbEvent.nTimestamp, fbGetTimeZoneInformation.tzInfo));
                aEventEntryTable[nEntryIndex].sTimestampCleared := SYSTEMTIME_TO_STRING(UlintToSystemTime(fbEvent.nTimestamp, fbGetTimeZoneInformation.tzInfo));

                aEventEntryTable[nEntryIndex].sTimestampCleared := SYSTEMTIME_TO_STRING(UlintToSystemTime(fbEvent.nTimestamp, fbGetTimeZoneInformation.tzInfo));
                stEventEntryTemp := aEventEntryTable[nEntryIndex];

                DeleteEntryFromEventTable(TO_UDINT(nEntryIndex));
            	nCounterNothingFound := 0;
			ELSE
				nCounterNothingFound := nCounterNothingFound + 1;
				IF nCounterNothingFound <= 20 THEN 
				bEventEntryTableTestandSet := FALSE;
				RETURN;	
				END_IF
				nCounterNothingFound := 0;
            END_IF
            
            stSeverestAlarmEntryTable:=  GetSeverestAlarmEntryTable();
            stLastEventEntryTable:=  GetLastEventEntryTable();
            UpdateLegacyTable(); 
            
            stEventEntryTemp.stAlarmLog.sTimestamp := stEventEntryTemp.sTimestampLog;      
            stEventEntryTemp.stAlarmLog.eConfirmationState := stEventEntryTemp.eConfirmationState;
            stEventEntryTemp.stAlarmLog.eSeverity := stEventEntryTemp.eSeverity;
            stEventEntryTemp.stAlarmLog.EventClassName := stEventEntryTemp.EventClassName;
            stEventEntryTemp.stAlarmLog.sSourceName := stEventEntryTemp.sSourceName;
            stEventEntryTemp.stAlarmLog.sText := stEventEntryTemp.sText;
            stEventEntryTemp.stAlarmLog.sTimestamp := REPLACE(STR1:= stEventEntryTemp.stAlarmLog.sTimestamp, STR2 := ' ',L := 1, P := 11);

            nStep := E_AlarmMessage.Done;

			bEventEntryTableTestandSet := FALSE;	
			END_IF	
	END_IF
    // CASE: Done   
    IF nStep = E_AlarmMessage.Done THEN  
            OnAlarmCleared := S_OK;
            nStep := E_AlarmMessage.RequestText;
            MEMSET(destAddr:= ADR(stEventEntryTemp), fillByte := 16#00 , n:= SIZEOF(stEventEntryTemp)); 
	END_IF     


// Fast Case of nStepRequestText
    // CASE: RequestText   
    IF nStepRequestText = E_AlarmMessage.RequestText THEN
        fbRequestText.Request(eventClass:=fbEvent.EventClass, nEventId:=fbEvent.nEventId, nLangId:=LangId, ipArgs:=fbEvent.ipArguments );
        nStepRequestText := E_AlarmMessage.ReceiveText; 
	END_IF
    // CASE: ReceiveText   
    IF nStepRequestText = E_AlarmMessage.ReceiveText THEN
        IF NOT fbRequestText.bBusy AND NOT fbRequestText.bError THEN
            fbRequestText.GetString(UTF8, SIZEOF(UTF8));
            UTF8_TO_STRING(pDstSTRING:=ADR(stEventEntryTemp.sText) , pSrcUTF8:=ADR(UTF8) , nDstSize:=SIZEOF(stEventEntryTemp.sText) , nDstLen=> );
            nStepRequestText := E_AlarmMessage.Done;
        ELSIF fbRequestText.bError THEN 
            nStepRequestText := E_AlarmMessage.RequestText;
        END_IF 
	END_IF
 
// Fast Case of nStepRequestClass
    // CASE: RequestText   
    IF nStepRequestClass = E_AlarmMessage.RequestText THEN
        fbRequestClassName.Request(eventClass:=fbEvent.EventClass, nLangId:=LangId,);
        nStepRequestClass := E_AlarmMessage.ReceiveText;
	END_IF
    // CASE: ReceiveText   
    IF nStepRequestClass = E_AlarmMessage.ReceiveText THEN
        IF NOT fbRequestClassName.bBusy AND NOT fbRequestClassName.bError THEN
            fbRequestClassName.GetString(UTF8, SIZEOF(UTF8));
            UTF8_TO_STRING(pDstSTRING:=ADR(stEventEntryTemp.EventClassName) , pSrcUTF8:=ADR(UTF8) , nDstSize:=SIZEOF(stEventEntryTemp.EventClassName) , nDstLen=> );
            nStepRequestClass := E_AlarmMessage.Done;
        ELSIF fbRequestClassName.bError THEN 
            nStepRequestClass := E_AlarmMessage.RequestText;
        END_IF
	END_IF
END_METHOD

METHOD OnAlarmConfirmed : HRESULT
VAR_INPUT
	fbEvent : REFERENCE TO FB_TcEvent;
END_VAR
VAR
    hr : HRESULT;
    UTF8 : STRING(255);
END_VAR
VAR_INST
    {attribute 'no_copy'}
    fbRequestText : FB_RequestEventText;
    {attribute 'no_copy'}
    fbRequestClassName : FB_RequestEventClassName;
	
	nCounterNothingFound : DINT;
END_VAR
VAR_INST
    stEventEntryTemp: ST_EventEntryTableListener;
END_VAR
VAR_INST
    nStep : E_AlarmMessage;
    nStepRequestText : E_AlarmMessage := E_AlarmMessage.Done;
    nStepRequestClass : E_AlarmMessage := E_AlarmMessage.Done;
END_VAR
VAR
nConfirmEntryIndex : DINT;
END_VAR

IF NOT __ISVALIDREF(fbEvent) THEN
	RETURN;
ELSE
	OnAlarmConfirmed := E_FAIL; // in order to receive more callbacks (Set <> S_OK in order to cancel the callbacks for this program cycle.)
	IF bChangeLanguageInterlock THEN
		RETURN;
	END_IF    
END_IF

// Fast Case of nStep
// CASE: E_AlarmMessage.RequestText
IF nStep = E_AlarmMessage.RequestText THEN
	nStepRequestText := E_AlarmMessage.RequestText;
	nStepRequestClass := E_AlarmMessage.RequestText;
	nStep := E_AlarmMessage.ReceiveText;
END_IF

// CASE: E_AlarmMessage.ReceiveText
IF nStep = E_AlarmMessage.ReceiveText THEN
	IF nStepRequestText = E_AlarmMessage.Done AND
		nStepRequestClass = E_AlarmMessage.Done THEN
		nStep := E_AlarmMessage.Insert;
	END_IF
END_IF

